ABB RAPID module: ProgSide1.mod

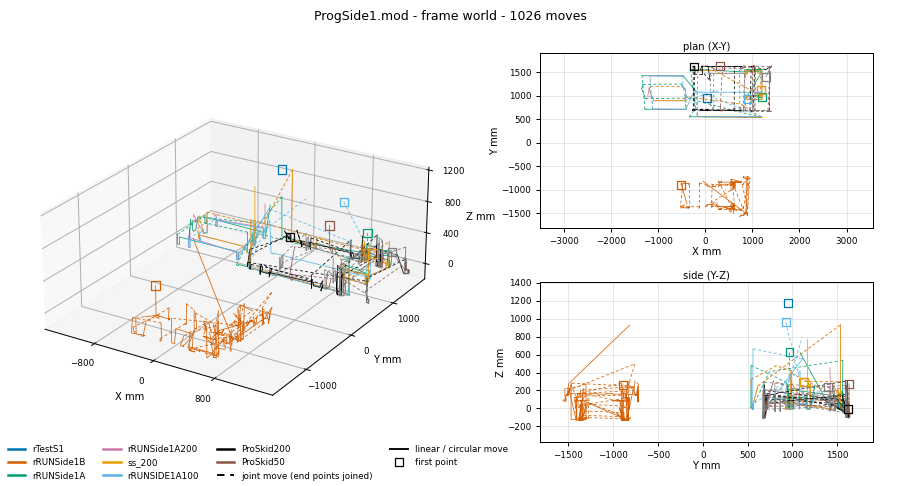
[picture p0: tool path of ProgSide1.mod in frame world, 1026 of 1039 moves have a stored position in this frame; points joined in program order, loops and branches not executed]
MODULE ProgSide1
	PERS bool bZ_B_onlySide2:=FALSE;
	PERS bool bZ_B_onlySide1:=FALSE;
	PERS bool bC_HalfstepSide2:=FALSE;
	PERS bool bC_HalfstepSide1:=FALSE;
	PERS bool bZ_HalfstepSide1:=FALSE;
	PERS bool bZ_HalfstepSide2:=FALSE;
	PERS bool bAngleSide1:=FALSE;
	PERS bool bAngleSide2:=FALSE;
	PERS bool bTestWeldSide1:=FALSE;
    PERS bool bTestWeldSide2:=FALSE;

    ! Boolian initialization for the SS 300 Frames
    PERS bool bNoPartSide1:=FALSE;
	PERS bool bNoPartSide2:=FALSE;
    PERS bool A_onlySide2:=FALSE;
    PERS bool B_onlySide2:=FALSE;
	PERS bool A_onlySide1:=FALSE;
    PERS bool B_onlySide1:=TRUE;
	PERS bool AB_Side1:=FALSE;
    PERS bool AB_Side2:=FALSE;

    ! Boolian initialization for the SelFrames procedures except the SS 300s.
    PERS bool bSkid50:=FALSE;
   	PERS bool bSkid100:=FALSE;
	PERS bool bSkid200:=FALSE;
    PERS bool bSide1A100:=FALSE;
    PERS bool bSide1A200:=FALSE;

    PERS bool bRover:=TRUE;


	TASK PERS welddata weld7:=[15.24,16.6963,[7,0,0,0,0,0,0,0,0],[7,0,0,0,0,0,0,0,0]];
	TASK PERS welddata weld6:=[16.2983,16.6963,[6,0,0,0,0,0,0,0,0],[6,0,0,0,0,0,0,0,0]];

	CONST robtarget pPounceOS1:=[[-398.58,690.45,580.22],[0.00101632,0.999968,-0.00455572,0.00645523],[-1,0,-1,0],[9E+09,9E+09,9E+09,9E+09,9E+09,9E+09]];
	CONST robtarget pPounceS21:=[[580.19,77.23,83.43],[0.071601,0.767336,-0.436334,0.464416],[-1,0,-2,0],[9E+09,9E+09,9E+09,9E+09,9E+09,9E+09]];
	TASK PERS seamdata seam2:=[4,1,[1,0,52,74.0833,0,0,0,0,0],0,0,0,0,0,[1,0,48,0,0,0,0,0,0],0.01,0.1,[1,0,48,105.833,0,0,0,0,0],0,0,[0,0,0,0,0,0,0,0,0],1];
	TASK PERS seamdata seam10:=[4,1,[1,0,50,80.4333,0,0,0,0,0],0,0,0,0,0,[0,0,0,0,0,0,0,0,0],0.25,0.25,[1,0,50,38.1,0,0,0,0,0],0,0,[0,0,0,0,0,0,0,0,0],1];
	CONST robtarget pPounceS31:=[[358.52,159.10,437.93],[0.0181628,-0.398765,0.916866,0.00362624],[-2,0,-2,0],[9E+09,9E+09,9E+09,9E+09,9E+09,9E+09]];
	CONST robtarget pPounceS41:=[[193.25,136.11,113.74],[0.188325,0.84715,-0.195157,0.45693],[-1,-1,-2,0],[9E+09,9E+09,9E+09,9E+09,9E+09,9E+09]];
	PERS welddata weld11:=[13.5467,0,[1,0,50,84.6667,0,0,0,0,0],[0,0,0,0,0,0,0,0,0]];
	PERS welddata weld10:=[14.8167,0,[1,0,50,95.25,0,0,0,0,0],[0,0,0,0,0,0,0,0,0]];
	TASK PERS seamdata seam11:=[1,1,[1,0,50,84.6667,0,0,0,0,0],0,0,0,0,0,[0,0,0,0,0,0,0,0,0],0,0,[0,0,0,0,0,0,0,0,0],0,0,[0,0,0,0,0,0,0,0,0],0];
	TASK PERS seamdata seam12:=[1,1,[1,0,18.5,381,0,0,0,0,0],0,0,0,0,0,[0,0,0,0,0,0,0,0,0],0,0,[0,0,0,0,0,0,0,0,0],0,0,[0,0,0,0,0,0,0,0,0],0];
	TASK PERS seamdata seam13:=[1,1,[1,0,14,127,0,0,0,0,0],0,0,0,0,0,[0,0,0,0,0,0,0,0,0],0,0,[0,0,0,0,0,0,0,0,0],0,0,[0,0,0,0,0,0,0,0,0],0];
	PERS welddata weld12:=[13.97,0,[1,0,50,84.6667,0,0,0,0,0],[0,0,0,0,0,0,0,0,0]];
	PERS welddata weld13:=[6.90033,0,[1,0,20,100.753,0,0,0,0,0],[0,0,0,0,0,0,0,0,0]];
	CONST robtarget pSafeS11:=[[-996.19,963.00,488.78],[0.0459907,-0.688393,0.722625,0.0425673],[1,-1,1,0],[9E+09,9E+09,9E+09,9E+09,9E+09,9E+09]];
	CONST robtarget pSafeS21:=[[-996.19,963.00,488.76],[0.0459983,-0.688397,0.722622,0.0425559],[1,-1,1,0],[9E+09,9E+09,9E+09,9E+09,9E+09,9E+09]];
	CONST robtarget pSafeS31:=[[506.44,675.04,711.34],[0.0314656,-0.935633,0.203865,-0.286426],[0,0,-2,0],[9E+09,9E+09,9E+09,9E+09,9E+09,9E+09]];
	CONST robtarget pSafeS41:=[[488.47,1091.24,654.25],[0.0459806,-0.688392,0.722627,0.0425664],[0,0,-1,0],[9E+09,9E+09,9E+09,9E+09,9E+09,9E+09]];
	CONST robtarget pSafeS51:=[[528.23,1196.89,528.24],[0.224235,-0.753625,-0.525201,-0.325471],[0,-1,-3,0],[9E+09,9E+09,9E+09,9E+09,9E+09,9E+09]];
	CONST robtarget pSafeS61:=[[597.29,1295.03,43.37],[0.191334,-0.732058,-0.538062,-0.371444],[0,-1,-2,0],[9E+09,9E+09,9E+09,9E+09,9E+09,9E+09]];
	CONST robtarget pSafeS71:=[[542.66,1322.39,535.75],[0.223485,-0.764556,-0.487458,-0.357621],[0,-1,-2,0],[9E+09,9E+09,9E+09,9E+09,9E+09,9E+09]];
	CONST robtarget pSafeS81:=[[542.66,1322.38,535.76],[0.223484,-0.764558,-0.487457,-0.35762],[0,-1,-2,0],[9E+09,9E+09,9E+09,9E+09,9E+09,9E+09]];
	CONST robtarget pPounceS51:=[[15.28,993.81,754.75],[0.277209,0.263034,-0.848831,-0.365313],[0,0,0,0],[9E+09,9E+09,9E+09,9E+09,9E+09,9E+09]];
	CONST robtarget pPounceS61:=[[649.55,1131.56,389.19],[0.45355,-0.00505177,-0.879595,-0.143459],[0,0,0,0],[9E+09,9E+09,9E+09,9E+09,9E+09,9E+09]];
	TASK PERS seamdata seam3:=[1,1,[1,0,35,84.6667,0,0,0,0,0],0,0,0,0,0,[1,0,48,0,0,0,0,0,0],0.01,0.1,[1,0,48,105.833,0,0,0,0,0],0,0,[0,0,0,0,0,0,0,0,0],1];
	CONST robtarget pSafeS101:=[[572.94,23.46,738.68],[0.0502756,-0.467207,-0.815726,-0.337314],[0,0,0,0],[9E+09,9E+09,9E+09,9E+09,9E+09,9E+09]];
	CONST robtarget pSafeS111:=[[877.74,-1.14,1156.39],[0.00629855,0.0017594,0.999979,-0.000494623],[0,-1,0,0],[9E+09,9E+09,9E+09,9E+09,9E+09,9E+09]];
	CONST robtarget pSafeS121:=[[877.74,-1.14,1156.39],[0.00629925,0.00175887,0.999979,-0.000492925],[0,-1,0,0],[9E+09,9E+09,9E+09,9E+09,9E+09,9E+09]];
	CONST robtarget pSafeS131:=[[865.02,1139.54,-19.77],[0.144708,-0.274627,0.931028,0.191903],[0,-2,2,0],[9E+09,9E+09,9E+09,9E+09,9E+09,9E+09]];
	CONST robtarget pSafeS141:=[[849.60,1148.97,-24.06],[0.00628216,0.00187497,0.999979,-0.000396021],[0,-1,1,0],[9E+09,9E+09,9E+09,9E+09,9E+09,9E+09]];
	CONST robtarget pSafeS151:=[[1007.97,1505.52,122.27],[0.0460025,-0.688387,0.722632,0.0425454],[0,1,-2,0],[9E+09,9E+09,9E+09,9E+09,9E+09,9E+09]];
	CONST robtarget pHomePos20:=[[365.14,988.92,-33.91],[0.0351389,-0.509982,-0.859022,-0.0276858],[0,-1,1,0],[9E+09,9E+09,9E+09,9E+09,9E+09,9E+09]];
	CONST robtarget pHomePos30:=[[365.15,979.87,-33.91],[0.0351433,-0.509968,-0.85903,-0.0276827],[0,-1,1,0],[9E+09,9E+09,9E+09,9E+09,9E+09,9E+09]];
	CONST robtarget pHomePos40:=[[365.14,979.87,-15.16],[0.0351385,-0.509986,-0.859019,-0.0276867],[0,-1,1,0],[9E+09,9E+09,9E+09,9E+09,9E+09,9E+09]];
	CONST robtarget pHomePos50:=[[433.12,979.73,-15.17],[0.0351369,-0.509964,-0.859032,-0.0276871],[0,-1,1,0],[9E+09,9E+09,9E+09,9E+09,9E+09,9E+09]];
	CONST robtarget pHomePos60:=[[430.57,978.47,-32.25],[0.0351433,-0.50998,-0.859023,-0.0276796],[0,-1,1,0],[9E+09,9E+09,9E+09,9E+09,9E+09,9E+09]];
	CONST robtarget pHomePos70:=[[430.57,978.46,-32.26],[0.0351393,-0.509989,-0.859017,-0.027681],[0,-1,1,0],[9E+09,9E+09,9E+09,9E+09,9E+09,9E+09]];
	CONST robtarget pHomePos80:=[[430.59,974.37,-32.26],[0.0351321,-0.50997,-0.859029,-0.0276862],[0,-1,1,0],[9E+09,9E+09,9E+09,9E+09,9E+09,9E+09]];
	CONST robtarget pHomePos90:=[[430.57,974.36,-24.94],[0.0351397,-0.509992,-0.859016,-0.0276799],[0,-1,1,0],[9E+09,9E+09,9E+09,9E+09,9E+09,9E+09]];
	CONST robtarget pHomePos100:=[[445.83,974.38,-24.94],[0.0351383,-0.509986,-0.859019,-0.0276863],[0,-1,1,0],[9E+09,9E+09,9E+09,9E+09,9E+09,9E+09]];
	CONST robtarget pHomePos110:=[[446.40,974.36,-32.29],[0.0351532,-0.510006,-0.859007,-0.0276708],[0,-1,1,0],[9E+09,9E+09,9E+09,9E+09,9E+09,9E+09]];
	CONST robtarget pHomePos120:=[[446.42,974.37,-32.29],[0.0351424,-0.509994,-0.859014,-0.0276814],[0,-1,1,0],[9E+09,9E+09,9E+09,9E+09,9E+09,9E+09]];
	CONST robtarget pSafeS12:=[[1424.79,-683.57,-13.74],[0.019551,0.168491,0.985501,-0.00412114],[-1,1,-2,0],[9E+09,9E+09,9E+09,9E+09,9E+09,9E+09]];
	CONST robtarget pSafeS22:=[[1462.93,-789.47,-110.40],[0.0637154,0.393325,0.863983,0.307846],[-1,1,-2,0],[9E+09,9E+09,9E+09,9E+09,9E+09,9E+09]];
	CONST robtarget pSafeS32:=[[1462.93,-821.54,-110.39],[0.0637158,0.39332,0.863986,0.307843],[-1,1,-2,0],[9E+09,9E+09,9E+09,9E+09,9E+09,9E+09]];
	CONST robtarget pSafeS42:=[[1462.93,-821.54,-110.39],[0.0637186,0.393326,0.863982,0.307849],[-1,1,-2,0],[9E+09,9E+09,9E+09,9E+09,9E+09,9E+09]];
	CONST robtarget pSafeS52:=[[1462.55,-1477.98,-107.56],[0.0637139,0.393324,0.863983,0.30785],[-1,0,-1,0],[9E+09,9E+09,9E+09,9E+09,9E+09,9E+09]];
	CONST robtarget pSafeS62:=[[1462.54,-1515.56,-107.57],[0.0637098,0.393325,0.863984,0.307846],[-1,0,-1,0],[9E+09,9E+09,9E+09,9E+09,9E+09,9E+09]];
	CONST robtarget pSafeS72:=[[1462.54,-1515.57,-107.57],[0.0637139,0.39333,0.86398,0.307849],[-1,0,-1,0],[9E+09,9E+09,9E+09,9E+09,9E+09,9E+09]];
	CONST robtarget pSafeS82:=[[1462.55,-1515.57,-6.77],[0.063723,0.393334,0.863975,0.307857],[-1,0,-1,0],[9E+09,9E+09,9E+09,9E+09,9E+09,9E+09]];
	CONST robtarget pSafeS161:=[[44.14,948.66,1172.82],[0.0459836,-0.688397,0.722622,0.0425714],[0,-1,0,0],[9E+09,9E+09,9E+09,9E+09,9E+09,9E+09]];
	CONST robtarget pSafeS171:=[[877.68,-1.12,1156.34],[0.00623811,0.00177345,0.999979,-0.000467886],[0,-1,0,0],[9E+09,9E+09,9E+09,9E+09,9E+09,9E+09]];
	CONST robtarget pSafeS181:=[[1178.99,1129.25,299.25],[0.0635535,0.517233,-0.779104,0.348467],[0,1,-3,1],[9E+09,9E+09,9E+09,9E+09,9E+09,9E+09]];
	CONST robtarget pSafeS191:=[[877.68,-1.12,1156.34],[0.00623811,0.00177268,0.999979,-0.000467882],[0,-1,0,0],[9E+09,9E+09,9E+09,9E+09,9E+09,9E+09]];
	CONST robtarget pSafeS201:=[[631.06,-50.80,790.98],[0.377429,-0.0153459,-0.925903,0.00402947],[-1,-1,-5,0],[9E+09,9E+09,9E+09,9E+09,9E+09,9E+09]];
	CONST robtarget pSafeS211:=[[631.06,-50.80,790.98],[0.377429,-0.0153486,-0.925903,0.00403031],[-1,-1,-5,0],[9E+09,9E+09,9E+09,9E+09,9E+09,9E+09]];


!XXXXXXXXXXXXXXXXXXXXXXXXXXXXXXXXXXXXXXXXXXXXXXXXXXXXXXXXXXXX

!XXXXXXXXXXXXXXXXXXXXXXXXXXXXXXXXXXXXXXXXXXXXXXXXXXXXXXXXXXXX
!xxxxxxxxxxxxxxxxxxxxxxxxxxxxxxxxxxxxxxxxxxxxxxxxxxxxxxxxxxxxxxxx




	PROC rNoPartS1()
		MoveJ pSafeS1, v800, fine, tWeldGun;
		MoveJ pPounceS1, v800, fine, tWeldGun;
		MoveJ pSafeS1, v800, fine, tWeldGun;
	ENDPROC
	PROC rTstA1()
		TPWrite "A S1";
	ENDPROC
	PROC rTstB1()
		TPWrite "B S1";
	ENDPROC
	PROC rTestS1()
		MoveJ [[44.14,948.66,1172.81],[0.0459874,-0.688394,0.722625,0.042569],[0,-1,0,0],[9E+09,9E+09,9E+09,9E+09,9E+09,9E+09]], v1000, z50, tWeldGun;
	ENDPROC
	PROC rRUNSide1B()
		rTestPosTop;
		TPWrite "Side 1 B";
		MoveJ [[-516.56,-891.88,262.76],[0.200577,-0.67934,-0.672798,-0.213563],[-2,0,-1,0],[9E+09,9E+09,9E+09,9E+09,9E+09,9E+09]], vmax, z10, tWeldGun;
		MoveL [[-517.38,-892.62,-126.02],[0.230166,-0.665805,-0.672085,-0.228101],[-2,0,-1,0],[9E+09,9E+09,9E+09,9E+09,9E+09,9E+09]], vmax, z10, tWeldGun;
		ArcLStart [[-517.38,-892.61,-138.56],[0.230168,-0.665801,-0.672089,-0.228098],[-2,0,-1,0],[9E+09,9E+09,9E+09,9E+09,9E+09,9E+09]], v50, seam13, weld13\Weave:=weave1, fine, tWeldGun;
		ArcLEnd [[-476.92,-892.72,-138.98],[0.230189,-0.665788,-0.672096,-0.228095],[-2,0,-1,0],[9E+09,9E+09,9E+09,9E+09,9E+09,9E+09]], v10, seam13, weld13\Weave:=weave1, fine, tWeldGun;
		MoveL [[-479.64,-891.87,-91.90],[0.200495,-0.679391,-0.672743,-0.213649],[-2,0,-1,0],[9E+09,9E+09,9E+09,9E+09,9E+09,9E+09]], vmax, z10, tWeldGun;
		MoveJ [[-526.59,-1340.74,-77.97],[0.272049,0.539222,-0.749573,0.270868],[-2,0,-3,0],[9E+09,9E+09,9E+09,9E+09,9E+09,9E+09]], vmax, z10, tWeldGun;
		MoveL [[-521.14,-1337.42,-124.98],[0.179758,0.684801,-0.680481,0.188893],[-2,-1,-3,0],[9E+09,9E+09,9E+09,9E+09,9E+09,9E+09]], vmax, z10, tWeldGun;
		ArcLStart [[-521.16,-1338.85,-130.75],[0.17975,0.684814,-0.680473,0.188882],[-2,-1,-3,0],[9E+09,9E+09,9E+09,9E+09,9E+09,9E+09]], v50, seam13, weld13\Weave:=weave1, fine, tWeldGun;
		ArcLEnd [[-484.70,-1342.96,-133.79],[0.179944,0.684785,-0.680418,0.189003],[-2,-1,-3,0],[9E+09,9E+09,9E+09,9E+09,9E+09,9E+09]], v10, seam13, weld13\Weave:=weave1, fine, tWeldGun;
		MoveL [[-484.84,-1342.71,46.50],[0.235633,0.655478,-0.679432,0.230648],[-2,-1,-3,0],[9E+09,9E+09,9E+09,9E+09,9E+09,9E+09]], vmax, z10, tWeldGun;
		MoveJ [[-392.56,-1296.67,69.52],[0.264192,0.731229,-0.303703,0.550702],[-2,0,0,0],[9E+09,9E+09,9E+09,9E+09,9E+09,9E+09]], vmax, z20, tWeldGun;
		MoveL [[-515.17,-856.60,-124.69],[0.238873,-0.653058,-0.67368,-0.250222],[-2,0,-1,0],[9E+09,9E+09,9E+09,9E+09,9E+09,9E+09]], vmax, z10, tWeldGun;
		ArcLStart [[-515.25,-854.21,-136.09],[0.220515,-0.671496,-0.67216,-0.220606],[-2,0,-1,0],[9E+09,9E+09,9E+09,9E+09,9E+09,9E+09]], v50, seam13, weld13, fine, tWeldGun;
		ArcLEnd [[-491.63,-854.12,-136.10],[0.220508,-0.671473,-0.67215,-0.220715],[-2,0,-1,0],[9E+09,9E+09,9E+09,9E+09,9E+09,9E+09]], v10, seam13, weld13\Weave:=weave1, fine, tWeldGun;
		MoveL [[-479.17,-861.28,-125.34],[0.171406,-0.677441,-0.683701,-0.210352],[-2,0,-1,0],[9E+09,9E+09,9E+09,9E+09,9E+09,9E+09]], vmax, z10, tWeldGun;
		MoveL [[-449.80,-861.68,-125.35],[0.171396,-0.677467,-0.683674,-0.21036],[-2,0,-1,0],[9E+09,9E+09,9E+09,9E+09,9E+09,9E+09]], vmax, z10, tWeldGun;
		ArcLStart [[-449.78,-856.11,-135.93],[0.208269,-0.667838,-0.686513,-0.198285],[-2,0,-1,0],[9E+09,9E+09,9E+09,9E+09,9E+09,9E+09]], v50, seam13, weld13\Weave:=weave1, fine, tWeldGun;
		ArcLEnd [[-419.12,-855.94,-135.97],[0.208222,-0.667816,-0.686496,-0.19847],[-2,0,-1,0],[9E+09,9E+09,9E+09,9E+09,9E+09,9E+09]], v10, seam13, weld13\Weave:=weave1, fine, tWeldGun;
		MoveL [[-410.60,-862.00,-128.92],[0.171386,-0.677508,-0.683632,-0.210375],[-2,0,-1,0],[9E+09,9E+09,9E+09,9E+09,9E+09,9E+09]], vmax, z10, tWeldGun;
		MoveL [[-376.40,-861.00,-128.93],[0.171385,-0.677516,-0.683626,-0.210371],[-2,0,-1,0],[9E+09,9E+09,9E+09,9E+09,9E+09,9E+09]], vmax, z10, tWeldGun;
		ArcLStart [[-376.97,-857.17,-135.72],[0.228827,-0.659649,-0.695979,-0.167674],[-2,0,-1,0],[9E+09,9E+09,9E+09,9E+09,9E+09,9E+09]], v50, seam13, weld13\Weave:=weave1, fine, tWeldGun;
		ArcLEnd [[-359.77,-857.10,-135.74],[0.228871,-0.659593,-0.696016,-0.167683],[-2,0,-1,0],[9E+09,9E+09,9E+09,9E+09,9E+09,9E+09]], v10, seam13, weld13\Weave:=weave1, fine, tWeldGun;
		MoveL [[-340.47,-873.25,-110.32],[0.171334,-0.677678,-0.683442,-0.210489],[-2,0,-1,0],[9E+09,9E+09,9E+09,9E+09,9E+09,9E+09]], vmax, z10, tWeldGun;
		!MoveJ [[-345.72,-887.43,-115.42],[0.0676146,-0.661673,-0.620705,-0.415143],[-2,0,-1,0],[9E+09,9E+09,9E+09,9E+09,9E+09,9E+09]], vmax, z10, tWeldGun;
		!MoveL [[-322.60,-865.30,-126.49],[0.067604,-0.661652,-0.620714,-0.415164],[-2,0,-1,0],[9E+09,9E+09,9E+09,9E+09,9E+09,9E+09]], vmax, z10, tWeldGun;
		!ArcLStart [[-323.53,-854.81,-126.59],[0.0676064,-0.661658,-0.620722,-0.415143],[-2,0,-1,0],[9E+09,9E+09,9E+09,9E+09,9E+09,9E+09]], v50, seam13, weld13, fine, tWeldGun;
		!ArcLEnd [[-310.94,-855.73,-127.27],[0.0675903,-0.661679,-0.620697,-0.415148],[-2,0,-1,0],[9E+09,9E+09,9E+09,9E+09,9E+09,9E+09]], v10, seam13, weld13, fine, tWeldGun;
		MoveL [[-354.07,-859.41,-129.42],[0.135806,-0.859729,-0.404621,-0.280545],[-2,-1,0,0],[9E+09,9E+09,9E+09,9E+09,9E+09,9E+09]], v100, z10, tWeldGun;
		ArcLStart [[-355.40,-857.25,-133.26],[0.101564,-0.865155,-0.372617,-0.319921],[-2,0,0,0],[9E+09,9E+09,9E+09,9E+09,9E+09,9E+09]], v10, seam13, weld13\Weave:=weave1, fine, tWeldGun;
		ArcLEnd [[-352.88,-886.23,-133.63],[0.0471147,-0.867186,-0.374018,-0.325392],[-2,0,-1,0],[9E+09,9E+09,9E+09,9E+09,9E+09,9E+09]], v10, seam13, weld13\Weave:=weave1, fine, tWeldGun;
		MoveL [[-337.59,-890.13,27.38],[0.0676709,-0.661709,-0.620708,-0.415072],[-2,0,-1,0],[9E+09,9E+09,9E+09,9E+09,9E+09,9E+09]], vmax, z10, tWeldGun;
		MoveJ [[-332.34,-1363.85,48.88],[0.219066,0.836756,-0.390875,0.31475],[-2,-1,1,0],[9E+09,9E+09,9E+09,9E+09,9E+09,9E+09]], vmax, z10, tWeldGun;
		MoveL [[-363.40,-1379.69,-125.19],[0.219062,0.836755,-0.390865,0.314767],[-2,-1,1,0],[9E+09,9E+09,9E+09,9E+09,9E+09,9E+09]], vmax, z10, tWeldGun;
		ArcLStart [[-360.34,-1385.64,-128.22],[0.219027,0.836785,-0.39084,0.314741],[-2,-1,1,0],[9E+09,9E+09,9E+09,9E+09,9E+09,9E+09]], v50, seam13, weld13\Weave:=weave1, fine, tWeldGun;
		ArcLEnd [[-360.74,-1353.82,-130.03],[0.219006,0.836811,-0.390806,0.314731],[-2,-1,1,0],[9E+09,9E+09,9E+09,9E+09,9E+09,9E+09]], v10, seam13, weld13\Weave:=weave1, fine, tWeldGun;
		MoveL [[-339.52,-1381.52,-122.91],[0.192161,0.836468,-0.399943,0.321625],[-2,-1,1,0],[9E+09,9E+09,9E+09,9E+09,9E+09,9E+09]], vmax, z10, tWeldGun;
		MoveL [[-360.99,-1380.78,-119.54],[0.218983,0.836818,-0.390808,0.314725],[-2,-1,1,0],[9E+09,9E+09,9E+09,9E+09,9E+09,9E+09]], vmax, z10, tWeldGun;
		ArcLStart [[-361.02,-1385.20,-130.65],[0.211582,0.836718,-0.393407,0.316807],[-2,-1,1,0],[9E+09,9E+09,9E+09,9E+09,9E+09,9E+09]], v10, seam13, weld13\Weave:=weave1, fine, tWeldGun;
		ArcLEnd [[-390.01,-1385.18,-131.66],[0.209306,0.844003,-0.389899,0.303035],[-2,-1,1,0],[9E+09,9E+09,9E+09,9E+09,9E+09,9E+09]], v10, seam13, weld13\Weave:=weave1, fine, tWeldGun;
		MoveL [[-390.07,-1379.88,-124.94],[0.206619,0.84095,-0.396616,0.304645],[-2,-1,1,0],[9E+09,9E+09,9E+09,9E+09,9E+09,9E+09]], vmax, z10, tWeldGun;
		!ArcLStart [[-352.45,-1380.36,-127.77],[0.213181,0.666131,-0.683648,0.208447],[-2,-1,1,0],[9E+09,9E+09,9E+09,9E+09,9E+09,9E+09]], v30, seam13, weld13, fine, tWeldGun;
		!ArcLEnd [[-392.89,-1382.82,-132.94],[0.213455,0.666087,-0.683527,0.208703],[-2,-1,1,0],[9E+09,9E+09,9E+09,9E+09,9E+09,9E+09]], v10, seam13, weld13, fine, tWeldGun;
		MoveL [[-383.12,-1377.19,-116.87],[0.247825,0.654497,-0.670463,0.246367],[-2,-1,1,0],[9E+09,9E+09,9E+09,9E+09,9E+09,9E+09]], vmax, z10, tWeldGun;
		MoveL [[-423.74,-1380.30,-127.27],[0.236796,0.658364,-0.678163,0.2249],[-2,-1,1,0],[9E+09,9E+09,9E+09,9E+09,9E+09,9E+09]], vmax, z10, tWeldGun;
		ArcLStart [[-423.76,-1381.10,-131.68],[0.205145,0.668814,-0.684061,0.206555],[-2,-1,1,0],[9E+09,9E+09,9E+09,9E+09,9E+09,9E+09]], v50, seam13, weld13\Weave:=weave1, fine, tWeldGun;
		ArcLEnd [[-450.34,-1381.29,-131.68],[0.205213,0.668788,-0.684058,0.206581],[-2,-1,1,0],[9E+09,9E+09,9E+09,9E+09,9E+09,9E+09]], v10, seam13, weld13\Weave:=weave1, fine, tWeldGun;
		MoveL [[-450.89,-1376.20,-127.31],[0.205227,0.668769,-0.684078,0.20656],[-2,-1,1,0],[9E+09,9E+09,9E+09,9E+09,9E+09,9E+09]], vmax, z10, tWeldGun;
		MoveL [[-485.27,-1373.50,-126.43],[0.24151,0.665828,-0.67086,0.219756],[-2,-1,1,0],[9E+09,9E+09,9E+09,9E+09,9E+09,9E+09]], vmax, z10, tWeldGun;
		ArcLStart [[-485.09,-1381.68,-132.22],[0.234587,0.663654,-0.676661,0.216014],[-2,-1,1,0],[9E+09,9E+09,9E+09,9E+09,9E+09,9E+09]], v50, seam13, weld13\Weave:=weave1, fine, tWeldGun;
		ArcLEnd [[-523.10,-1381.58,-132.24],[0.234599,0.66365,-0.676663,0.216008],[-2,-1,1,0],[9E+09,9E+09,9E+09,9E+09,9E+09,9E+09]], v10, seam13, weld13\Weave:=weave1, fine, tWeldGun;
		MoveL [[-522.10,-1355.74,48.22],[0.158867,0.68146,-0.647455,0.301955],[-2,0,1,0],[9E+09,9E+09,9E+09,9E+09,9E+09,9E+09]], vmax, z10, tWeldGun;
		MoveJ [[-133.27,-1356.80,81.68],[0.311551,0.028851,-0.949681,-0.0145225],[-2,0,-2,0],[9E+09,9E+09,9E+09,9E+09,9E+09,9E+09]], vmax, z10, tWeldGun;
		MoveL [[-129.77,-1359.47,-118.55],[0.313406,-0.0329684,-0.948479,0.032837],[-2,0,-2,0],[9E+09,9E+09,9E+09,9E+09,9E+09,9E+09]], vmax, z10, tWeldGun;
		ArcLStart [[-130.10,-1360.61,-131.11],[0.319988,-0.0412281,-0.946509,0.00534418],[-2,0,-2,0],[9E+09,9E+09,9E+09,9E+09,9E+09,9E+09]], v50, seam13, weld13\Weave:=weave1, fine, tWeldGun;
		ArcLEnd [[-130.29,-1389.82,-131.10],[0.320004,-0.0412218,-0.946504,0.00536126],[-2,0,-2,0],[9E+09,9E+09,9E+09,9E+09,9E+09,9E+09]], v10, seam13, weld13\Weave:=weave1, fine, tWeldGun;
		MoveL [[-127.94,-1387.70,-99.83],[0.311507,0.0288878,-0.94969,-0.0147574],[-2,0,-2,0],[9E+09,9E+09,9E+09,9E+09,9E+09,9E+09]], vmax, z10, tWeldGun;
		MoveJ [[-120.34,-878.23,-115.66],[0.321395,0.00587998,-0.946893,0.00807266],[-2,0,-2,0],[9E+09,9E+09,9E+09,9E+09,9E+09,9E+09]], vmax, z10, tWeldGun;
		MoveL [[-125.84,-880.54,-126.77],[0.319682,0.0182803,-0.947348,-0.00115479],[-2,0,-2,0],[9E+09,9E+09,9E+09,9E+09,9E+09,9E+09]], vmax, z10, tWeldGun;
		ArcLStart [[-127.17,-881.43,-133.73],[0.308264,0.0190236,-0.951103,0.00389985],[-2,0,-2,0],[9E+09,9E+09,9E+09,9E+09,9E+09,9E+09]], v50, seam13, weld13\Weave:=weave1, fine, tWeldGun;
		ArcLEnd [[-126.99,-850.35,-133.72],[0.308286,0.0190346,-0.951095,0.00390381],[-2,0,-2,0],[9E+09,9E+09,9E+09,9E+09,9E+09,9E+09]], v10, seam13, weld13\Weave:=weave1, fine, tWeldGun;
		MoveL [[-126.07,-851.54,117.21],[0.311664,0.0289025,-0.949643,-0.0144782],[-2,0,-2,0],[9E+09,9E+09,9E+09,9E+09,9E+09,9E+09]], vmax, z10, tWeldGun;
		MoveJ [[5.08,-892.16,87.65],[0.246917,-0.649526,-0.670091,-0.261011],[-2,0,-1,0],[9E+09,9E+09,9E+09,9E+09,9E+09,9E+09]], vmax, z10, tWeldGun;
		MoveL [[5.70,-898.13,-125.58],[0.246931,-0.64953,-0.670081,-0.261012],[-2,0,-1,0],[9E+09,9E+09,9E+09,9E+09,9E+09,9E+09]], vmax, z10, tWeldGun;
		ArcLStart [[8.01,-895.77,-137.58],[0.202938,-0.669252,-0.681328,-0.216127],[-2,0,-1,0],[9E+09,9E+09,9E+09,9E+09,9E+09,9E+09]], v50, seam13, weld13\Weave:=weave1, fine, tWeldGun;
		ArcLEnd [[39.00,-896.37,-138.18],[0.202954,-0.669237,-0.681341,-0.216117],[-1,0,-1,0],[9E+09,9E+09,9E+09,9E+09,9E+09,9E+09]], v10, seam13, weld13\Weave:=weave1, fine, tWeldGun;
		MoveL [[40.66,-920.62,70.48],[0.246699,-0.649617,-0.670207,-0.260692],[-1,0,-1,0],[9E+09,9E+09,9E+09,9E+09,9E+09,9E+09]], vmax, z10, tWeldGun;
		MoveJ [[283.83,-931.65,13.13],[0.246958,-0.649486,-0.670134,-0.26096],[-1,0,0,0],[9E+09,9E+09,9E+09,9E+09,9E+09,9E+09]], vmax, z10, tWeldGun;
		MoveL [[286.40,-898.85,-115.99],[0.246961,-0.649476,-0.670147,-0.26095],[-1,0,0,0],[9E+09,9E+09,9E+09,9E+09,9E+09,9E+09]], vmax, z10, tWeldGun;
		ArcLStart [[287.27,-897.40,-138.20],[0.199806,-0.665794,-0.68607,-0.214718],[-1,-1,0,0],[9E+09,9E+09,9E+09,9E+09,9E+09,9E+09]], v50, seam13, weld13\Weave:=weave1, fine, tWeldGun;
		ArcLEnd [[316.06,-898.20,-138.20],[0.19983,-0.665775,-0.686086,-0.214705],[-1,-1,0,0],[9E+09,9E+09,9E+09,9E+09,9E+09,9E+09]], v10, seam13, weld13\Weave:=weave1, fine, tWeldGun;
		MoveL [[299.75,-898.83,-116.82],[0.246966,-0.649478,-0.670145,-0.260945],[-1,0,0,0],[9E+09,9E+09,9E+09,9E+09,9E+09,9E+09]], vmax, z10, tWeldGun;
		MoveJ [[559.57,-898.83,-116.82],[0.246966,-0.649476,-0.670148,-0.260944],[-1,-1,0,0],[9E+09,9E+09,9E+09,9E+09,9E+09,9E+09]], vmax, z10, tWeldGun;
		MoveL [[564.80,-902.55,-126.00],[0.209407,-0.662689,-0.684007,-0.221648],[-1,-1,0,0],[9E+09,9E+09,9E+09,9E+09,9E+09,9E+09]], vmax, z10, tWeldGun;
		ArcLStart [[567.30,-900.67,-135.77],[0.209518,-0.662633,-0.684042,-0.221601],[-1,-1,0,0],[9E+09,9E+09,9E+09,9E+09,9E+09,9E+09]], v50, seam13, weld13\Weave:=weave1, fine, tWeldGun;
		ArcLEnd [[598.83,-900.83,-136.39],[0.209539,-0.662615,-0.684059,-0.221582],[-1,-1,0,0],[9E+09,9E+09,9E+09,9E+09,9E+09,9E+09]], v10, seam13, weld13\Weave:=weave1, fine, tWeldGun;
		MoveL [[596.75,-960.43,-56.34],[0.246991,-0.649449,-0.670174,-0.260919],[-1,-1,0,0],[9E+09,9E+09,9E+09,9E+09,9E+09,9E+09]], vmax, z10, tWeldGun;
		MoveJ [[601.90,-897.43,-123.32],[0.32616,-0.613254,-0.630335,-0.346725],[-1,0,0,0],[9E+09,9E+09,9E+09,9E+09,9E+09,9E+09]], vmax, z10, tWeldGun;
		MoveL [[600.91,-903.21,-128.01],[0.274675,-0.639039,-0.654325,-0.296719],[-1,0,0,0],[9E+09,9E+09,9E+09,9E+09,9E+09,9E+09]], v100, z10, tWeldGun;
		ArcLStart [[600.91,-897.21,-134.81],[0.274671,-0.63904,-0.654325,-0.296721],[-1,0,0,0],[9E+09,9E+09,9E+09,9E+09,9E+09,9E+09]], v10, seam13, weld13\Weave:=weave1, fine, tWeldGun;
		ArcLEnd [[631.68,-897.21,-134.82],[0.274687,-0.639035,-0.654325,-0.296718],[-1,0,0,0],[9E+09,9E+09,9E+09,9E+09,9E+09,9E+09]], v10, seam13, weld13\Weave:=weave1, fine, tWeldGun;
		MoveL [[633.74,-910.04,-132.93],[0.326202,-0.613258,-0.630325,-0.346695],[-1,0,0,0],[9E+09,9E+09,9E+09,9E+09,9E+09,9E+09]], vmax, z10, tWeldGun;
		MoveL [[633.73,-910.04,183.03],[0.326216,-0.613247,-0.630334,-0.346685],[-1,0,0,0],[9E+09,9E+09,9E+09,9E+09,9E+09,9E+09]], vmax, z10, tWeldGun;
		MoveJ [[627.00,-822.44,298.30],[0.361159,0.600904,-0.609737,0.36973],[-1,-1,-2,0],[9E+09,9E+09,9E+09,9E+09,9E+09,9E+09]], vmax, z10, tWeldGun;
		MoveL [[626.21,-835.86,-135.39],[0.402337,0.574507,-0.586331,0.405317],[-1,-2,-1,0],[9E+09,9E+09,9E+09,9E+09,9E+09,9E+09]], vmax, z10, tWeldGun;
		ArcLStart [[627.33,-853.89,-136.93],[0.402422,0.574444,-0.586338,0.405314],[-1,-2,-1,0],[9E+09,9E+09,9E+09,9E+09,9E+09,9E+09]], v50, seam13, weld13\Weave:=weave1, fine, tWeldGun;
		ArcLEnd [[595.13,-853.88,-136.75],[0.402409,0.574476,-0.586313,0.405318],[-1,-2,-1,0],[9E+09,9E+09,9E+09,9E+09,9E+09,9E+09]], v10, seam13, weld13\Weave:=weave1, fine, tWeldGun;
		MoveL [[595.98,-827.09,-135.34],[0.402393,0.574513,-0.586267,0.405347],[-1,-2,-1,0],[9E+09,9E+09,9E+09,9E+09,9E+09,9E+09]], vmax, z10, tWeldGun;
		MoveL [[626.55,-840.41,83.52],[0.487695,0.50329,-0.532941,0.47416],[-1,-2,-1,0],[9E+09,9E+09,9E+09,9E+09,9E+09,9E+09]], vmax, z10, tWeldGun;
		!MoveJ [[591.71,-1338.72,-121.22],[0.313919,0.593482,-0.705938,0.225579],[-1,-1,2,0],[9E+09,9E+09,9E+09,9E+09,9E+09,9E+09]], v1000, z10, tWeldGun;
		!MoveL [[591.71,-1350.59,-131.13],[0.31392,0.593478,-0.705939,0.225584],[-1,-1,2,0],[9E+09,9E+09,9E+09,9E+09,9E+09,9E+09]], v1000, z10, tWeldGun;
		ArcLStart [[627.59,-855.49,80.83],[0.48302,0.507656,-0.528665,0.479052],[-1,-2,-1,0],[9E+09,9E+09,9E+09,9E+09,9E+09,9E+09]], v40, seam13, weld13\Weave:=weave1, fine, tWeldGun;
		ArcLEnd [[594.18,-855.46,80.81],[0.483027,0.507675,-0.528656,0.479035],[-1,-2,-1,0],[9E+09,9E+09,9E+09,9E+09,9E+09,9E+09]], v10, seam13, weld13\Weave:=weave1, fine, tWeldGun;
		MoveL [[594.80,-840.42,83.53],[0.487698,0.503251,-0.532984,0.47415],[-1,-2,-1,0],[9E+09,9E+09,9E+09,9E+09,9E+09,9E+09]], vmax, z10, tWeldGun;
		SingArea\Wrist;
		MoveJ [[510.38,-859.01,160.69],[0.00485322,0.746032,-0.024255,0.665452],[-1,0,0,0],[9E+09,9E+09,9E+09,9E+09,9E+09,9E+09]], vmax, z10, tWeldGun;
		MoveL [[594.98,-857.13,82.26],[0.0048321,0.745919,-0.0242101,0.665579],[-1,0,0,0],[9E+09,9E+09,9E+09,9E+09,9E+09,9E+09]], vmax, z10, tWeldGun;
		ArcLStart [[600.76,-855.94,81.47],[0.00483992,0.74593,-0.0242017,0.665567],[-1,0,0,0],[9E+09,9E+09,9E+09,9E+09,9E+09,9E+09]], v40, seam13, weld13\Weave:=weave1, fine, tWeldGun;
		ArcLEnd [[600.72,-888.35,80.66],[0.00484822,0.745947,-0.0241951,0.665549],[-1,0,0,0],[9E+09,9E+09,9E+09,9E+09,9E+09,9E+09]], v10, seam13, weld13\Weave:=weave1, fine, tWeldGun;
		MoveL [[545.64,-889.59,83.73],[0.0047987,0.745982,-0.0242261,0.665508],[-1,0,0,0],[9E+09,9E+09,9E+09,9E+09,9E+09,9E+09]], vmax, z10, tWeldGun;
		MoveL [[545.47,-1007.73,83.69],[0.00477345,0.745999,-0.0242032,0.665491],[-1,0,0,0],[9E+09,9E+09,9E+09,9E+09,9E+09,9E+09]], vmax, z10, tWeldGun;
		MoveJ [[631.13,-962.99,83.64],[0.467638,-0.538268,-0.512971,-0.477958],[-1,0,0,0],[9E+09,9E+09,9E+09,9E+09,9E+09,9E+09]], vmax, z10, tWeldGun;
		MoveL [[598.81,-898.79,83.47],[0.467222,-0.531735,-0.519712,-0.478395],[-1,0,0,0],[9E+09,9E+09,9E+09,9E+09,9E+09,9E+09]], vmax, z10, tWeldGun;
		ArcLStart [[601.50,-884.14,82.85],[0.46721,-0.531727,-0.519721,-0.478406],[-1,0,0,0],[9E+09,9E+09,9E+09,9E+09,9E+09,9E+09]], v50, seam13, weld13\Weave:=weave1, fine, tWeldGun;
		ArcLEnd [[633.51,-883.86,83.69],[0.46722,-0.531721,-0.519715,-0.478409],[-1,0,0,0],[9E+09,9E+09,9E+09,9E+09,9E+09,9E+09]], v10, seam13, weld13\Weave:=weave1, fine, tWeldGun;
		MoveL [[633.84,-953.29,84.81],[0.467086,-0.531839,-0.51974,-0.478381],[-1,0,0,0],[9E+09,9E+09,9E+09,9E+09,9E+09,9E+09]], vmax, z10, tWeldGun;
		MoveJ [[-0.34,-1346.80,171.20],[0.287604,0.644423,-0.651566,0.278325],[-1,-1,-2,0],[9E+09,9E+09,9E+09,9E+09,9E+09,9E+09]], vmax, z10, tWeldGun;
		MoveL [[-2.12,-1347.00,-106.57],[0.287602,0.644471,-0.651521,0.278323],[-1,-1,-2,0],[9E+09,9E+09,9E+09,9E+09,9E+09,9E+09]], vmax, z10, tWeldGun;
		ArcLStart [[0.53,-1348.45,-134.66],[0.24536,0.661385,-0.66625,0.241826],[-1,0,-2,0],[9E+09,9E+09,9E+09,9E+09,9E+09,9E+09]], v40, seam13, weld13\Weave:=weave1, fine, tWeldGun;
		ArcLEnd [[35.28,-1348.02,-135.08],[0.245344,0.66148,-0.666161,0.241829],[-1,0,-2,0],[9E+09,9E+09,9E+09,9E+09,9E+09,9E+09]], v10, seam13, weld13\Weave:=weave1, fine, tWeldGun;
		MoveL [[33.45,-1306.76,35.10],[0.287609,0.644475,-0.651512,0.278328],[-1,-1,-2,0],[9E+09,9E+09,9E+09,9E+09,9E+09,9E+09]], vmax, z10, tWeldGun;
		MoveL [[273.41,-1327.02,35.12],[0.287608,0.6445,-0.651487,0.278327],[-1,-1,-2,0],[9E+09,9E+09,9E+09,9E+09,9E+09,9E+09]], vmax, z10, tWeldGun;
		MoveL [[278.63,-1350.36,-113.58],[0.287595,0.644518,-0.651477,0.278323],[-1,-1,-2,0],[9E+09,9E+09,9E+09,9E+09,9E+09,9E+09]], vmax, z10, tWeldGun;
		ArcLStart [[281.41,-1351.07,-135.11],[0.23791,0.664067,-0.669311,0.233317],[-1,0,-2,0],[9E+09,9E+09,9E+09,9E+09,9E+09,9E+09]], v40, seam13, weld13\Weave:=weave1, fine, tWeldGun;
		ArcLEnd [[314.07,-1351.40,-135.14],[0.237905,0.66408,-0.669298,0.233324],[-1,0,-2,0],[9E+09,9E+09,9E+09,9E+09,9E+09,9E+09]], v10, seam13, weld13\Weave:=weave1, fine, tWeldGun;
		MoveL [[313.56,-1350.36,-117.72],[0.287596,0.644518,-0.651477,0.278324],[-1,-1,-2,0],[9E+09,9E+09,9E+09,9E+09,9E+09,9E+09]], vmax, z10, tWeldGun;
		MoveL [[556.08,-1348.76,-117.74],[0.287601,0.644532,-0.651463,0.278317],[-1,-1,-2,0],[9E+09,9E+09,9E+09,9E+09,9E+09,9E+09]], vmax, z10, tWeldGun;
		ArcLStart [[558.44,-1352.44,-134.04],[0.243015,0.662361,-0.668163,0.23618],[-1,0,-2,0],[9E+09,9E+09,9E+09,9E+09,9E+09,9E+09]], v40, seam13, weld13\Weave:=weave1, fine, tWeldGun;
		ArcLEnd [[594.43,-1353.65,-134.07],[0.265401,0.653922,-0.658502,0.26139],[-1,0,-2,0],[9E+09,9E+09,9E+09,9E+09,9E+09,9E+09]], v10, seam13, weld13\Weave:=weave1, fine, tWeldGun;
		MoveL [[591.10,-1294.92,-96.48],[0.287644,0.644544,-0.6514,0.278391],[-1,-1,-2,0],[9E+09,9E+09,9E+09,9E+09,9E+09,9E+09]], vmax, z10, tWeldGun;
		!MoveJ [[629.17,-1265.05,-98.00],[0.340013,0.628245,-0.617658,0.328935],[-1,-1,-2,0],[9E+09,9E+09,9E+09,9E+09,9E+09,9E+09]], vmax, z10, tWeldGun;
		MoveL [[623.54,-1349.21,-127.64],[0.3277,0.635367,-0.623181,0.317123],[-1,-1,-2,0],[9E+09,9E+09,9E+09,9E+09,9E+09,9E+09]], vmax, z10, tWeldGun;
		ArcLStart [[622.97,-1358.18,-133.65],[0.327698,0.635371,-0.623176,0.317128],[-1,-1,-2,0],[9E+09,9E+09,9E+09,9E+09,9E+09,9E+09]], v40, seam13, weld13\Weave:=weave1, fine, tWeldGun;
		ArcLEnd [[591.94,-1357.90,-133.23],[0.327693,0.635344,-0.623186,0.317167],[-1,-1,-2,0],[9E+09,9E+09,9E+09,9E+09,9E+09,9E+09]], v10, seam13, weld13\Weave:=weave1, fine, tWeldGun;
		MoveL [[594.26,-1304.04,-124.90],[0.375061,0.603881,-0.605571,0.35769],[-1,-1,-2,0],[9E+09,9E+09,9E+09,9E+09,9E+09,9E+09]], vmax, z10, tWeldGun;
		MoveL [[594.27,-1304.02,270.29],[0.377187,0.607515,-0.60193,0.355439],[-1,-1,-2,0],[9E+09,9E+09,9E+09,9E+09,9E+09,9E+09]], vmax, z10, tWeldGun;
		MoveJ [[598.90,-1494.47,216.89],[0.17643,-0.701594,-0.668329,-0.173135],[-1,-1,0,0],[9E+09,9E+09,9E+09,9E+09,9E+09,9E+09]], vmax, z10, tWeldGun;
		MoveL [[597.76,-1413.70,-132.21],[0.38046,-0.610425,-0.582563,-0.378488],[-1,0,0,0],[9E+09,9E+09,9E+09,9E+09,9E+09,9E+09]], vmax, z10, tWeldGun;
		ArcLStart [[594.86,-1404.13,-132.25],[0.380476,-0.61045,-0.582552,-0.378447],[-1,0,0,0],[9E+09,9E+09,9E+09,9E+09,9E+09,9E+09]], v50, seam13, weld13\Weave:=weave1, fine, tWeldGun;
		ArcLEnd [[628.57,-1403.11,-132.15],[0.38049,-0.610453,-0.582547,-0.378435],[-1,0,0,0],[9E+09,9E+09,9E+09,9E+09,9E+09,9E+09]], v10, seam13, weld13\Weave:=weave1, fine, tWeldGun;
		MoveL [[628.36,-1412.35,-121.21],[0.467542,-0.524108,-0.539123,-0.464825],[-1,0,0,0],[9E+09,9E+09,9E+09,9E+09,9E+09,9E+09]], vmax, z10, tWeldGun;
		MoveL [[629.51,-1407.41,86.42],[0.467564,-0.524053,-0.539189,-0.464788],[-1,0,0,0],[9E+09,9E+09,9E+09,9E+09,9E+09,9E+09]], vmax, z10, tWeldGun;
		ArcLStart [[628.33,-1394.78,86.06],[0.467613,-0.524083,-0.539148,-0.464753],[-1,0,0,0],[9E+09,9E+09,9E+09,9E+09,9E+09,9E+09]], v40, seam13, weld13\Weave:=weave1, fine, tWeldGun;
		ArcLEnd [[594.53,-1394.77,86.03],[0.467622,-0.524085,-0.539138,-0.464753],[-1,0,0,0],[9E+09,9E+09,9E+09,9E+09,9E+09,9E+09]], v10, seam13, weld13\Weave:=weave1, fine, tWeldGun;
		MoveL [[595.96,-1403.58,86.03],[0.467592,-0.524062,-0.539124,-0.464825],[-1,0,0,0],[9E+09,9E+09,9E+09,9E+09,9E+09,9E+09]], vmax, z10, tWeldGun;
		MoveL [[457.06,-1403.59,89.42],[0.225264,-0.323777,-0.705869,-0.588366],[-1,0,-1,0],[9E+09,9E+09,9E+09,9E+09,9E+09,9E+09]], vmax, z10, tWeldGun;
		MoveJ [[483.55,-1400.78,96.25],[0.150969,0.719954,0.110873,0.668268],[-1,0,0,0],[9E+09,9E+09,9E+09,9E+09,9E+09,9E+09]], vmax, z10, tWeldGun;
		MoveL [[583.47,-1400.75,85.01],[0.0329721,0.73526,0.0213877,0.676645],[-1,0,0,0],[9E+09,9E+09,9E+09,9E+09,9E+09,9E+09]], vmax, z10, tWeldGun;
		ArcLStart [[594.01,-1399.37,84.43],[0.0288105,0.735302,0.0250795,0.676663],[-1,0,0,0],[9E+09,9E+09,9E+09,9E+09,9E+09,9E+09]], v50, seam13, weld13\Weave:=weave1, fine, tWeldGun;
		ArcLEnd [[593.57,-1367.91,84.17],[0.028766,0.73533,0.0251421,0.676632],[-1,0,0,0],[9E+09,9E+09,9E+09,9E+09,9E+09,9E+09]], v10, seam13, weld13\Weave:=weave1, fine, tWeldGun;
		MoveL [[554.18,-1372.28,89.73],[0.15109,0.720146,0.110407,0.668112],[-1,0,0,0],[9E+09,9E+09,9E+09,9E+09,9E+09,9E+09]], vmax, z10, tWeldGun;
		MoveL [[549.71,-1268.25,89.71],[0.151117,0.720151,0.110329,0.668113],[-1,1,0,0],[9E+09,9E+09,9E+09,9E+09,9E+09,9E+09]], vmax, z10, tWeldGun;
		MoveJ [[603.39,-1313.43,143.58],[0.469159,0.533622,-0.523436,0.470269],[-1,-2,3,0],[9E+09,9E+09,9E+09,9E+09,9E+09,9E+09]], vmax, z10, tWeldGun;
		MoveL [[591.28,-1347.97,82.12],[0.473675,0.523571,-0.526883,0.473181],[-1,-2,3,0],[9E+09,9E+09,9E+09,9E+09,9E+09,9E+09]], vmax, z10, tWeldGun;
		ArcLStart [[587.84,-1367.93,83.28],[0.473679,0.523503,-0.526973,0.473152],[-1,-2,3,0],[9E+09,9E+09,9E+09,9E+09,9E+09,9E+09]], v40, seam13, weld13\Weave:=weave1, fine, tWeldGun;
		ArcLEnd [[621.99,-1367.50,82.25],[0.473695,0.523434,-0.527058,0.473118],[-1,-2,3,0],[9E+09,9E+09,9E+09,9E+09,9E+09,9E+09]], v10, seam13, weld13\Weave:=weave1, fine, tWeldGun;
		MoveL [[621.57,-1338.36,83.93],[0.473691,0.523533,-0.526918,0.473168],[-1,-2,3,0],[9E+09,9E+09,9E+09,9E+09,9E+09,9E+09]], vmax, z10, tWeldGun;
		!MoveL [[592.94,-1347.68,-124.63],[0.145068,0.695314,-0.634216,0.305394],[-1,0,1,0],[9E+09,9E+09,9E+09,9E+09,9E+09,9E+09]], vmax, z10, tWeldGun;
		!ArcLStart [[592.95,-1351.62,-131.66],[0.121904,0.705948,-0.639076,0.279928],[-1,0,1,0],[9E+09,9E+09,9E+09,9E+09,9E+09,9E+09]], v40, seam13, weld13\Weave:=weave1, fine, tWeldGun;
		!ArcLEnd [[553.63,-1351.63,-131.65],[0.121904,0.705942,-0.639079,0.279934],[-1,0,1,0],[9E+09,9E+09,9E+09,9E+09,9E+09,9E+09]], v10, seam13, weld13\Weave:=weave1, fine, tWeldGun;
		!MoveL [[558.95,-1354.44,-113.35],[0.145045,0.695254,-0.634278,0.305412],[-1,0,1,0],[9E+09,9E+09,9E+09,9E+09,9E+09,9E+09]], vmax, z10, tWeldGun;
		!MoveL [[313.92,-1351.24,-119.86],[0.226173,0.673271,-0.665892,0.228343],[-1,0,2,0],[9E+09,9E+09,9E+09,9E+09,9E+09,9E+09]], vmax, z10, tWeldGun;
		!ArcLStart [[315.31,-1349.16,-136.09],[0.226124,0.673334,-0.665847,0.228338],[-1,0,2,0],[9E+09,9E+09,9E+09,9E+09,9E+09,9E+09]], v40, seam13, weld13\Weave:=weave1, fine, tWeldGun;
		!ArcLEnd [[277.70,-1348.77,-134.69],[0.226134,0.673338,-0.66584,0.228336],[-1,0,2,0],[9E+09,9E+09,9E+09,9E+09,9E+09,9E+09]], v10, seam13, weld13\Weave:=weave1, fine, tWeldGun;
		!MoveL [[279.11,-1351.10,-105.85],[0.22616,0.673298,-0.665876,0.228321],[-1,0,2,0],[9E+09,9E+09,9E+09,9E+09,9E+09,9E+09]], vmax, z10, tWeldGun;
		MoveJ [[584.48,-948.55,-60.93],[0.252385,-0.649774,-0.664987,-0.268121],[-1,0,0,0],[9E+09,9E+09,9E+09,9E+09,9E+09,9E+09]], vmax, z10, tWeldGun;
		MoveL [[587.25,-889.04,-107.33],[0.252799,-0.649451,-0.665162,-0.268079],[-1,0,0,0],[9E+09,9E+09,9E+09,9E+09,9E+09,9E+09]], vmax, z10, tWeldGun;
		ArcLStart [[587.97,-882.93,-130.55],[0.253029,-0.649357,-0.665187,-0.268027],[-1,0,0,0],[9E+09,9E+09,9E+09,9E+09,9E+09,9E+09]], v40, seam13, weld13\Weave:=weave1, fine, tWeldGun;
		ArcL [[579.89,-891.69,-131.98],[0.25302,-0.649426,-0.665094,-0.2681],[-1,0,0,0],[9E+09,9E+09,9E+09,9E+09,9E+09,9E+09]], v10, seam13, weld13\Weave:=weave1, z0, tWeldGun;
		ArcL [[479.92,-890.95,-132.98],[0.253042,-0.649377,-0.665146,-0.26807],[-1,0,0,0],[9E+09,9E+09,9E+09,9E+09,9E+09,9E+09]], v10, seam13, weld13\Weave:=weave1, z0, tWeldGun;
		ArcLEnd [[469.00,-879.31,-133.61],[0.253095,-0.649334,-0.665183,-0.26803],[-1,0,0,0],[9E+09,9E+09,9E+09,9E+09,9E+09,9E+09]], v10, seam13, weld13\Weave:=weave1, fine, tWeldGun;
		MoveL [[472.59,-879.09,-111.98],[0.253025,-0.6494,-0.665124,-0.268085],[-1,0,0,0],[9E+09,9E+09,9E+09,9E+09,9E+09,9E+09]], vmax, z10, tWeldGun;
		MoveL [[396.83,-879.33,-105.08],[0.253072,-0.649383,-0.665131,-0.268064],[-1,0,0,0],[9E+09,9E+09,9E+09,9E+09,9E+09,9E+09]], vmax, z10, tWeldGun;
		ArcLStart [[396.64,-879.58,-133.89],[0.25962,-0.646746,-0.667845,-0.261344],[-1,-1,0,0],[9E+09,9E+09,9E+09,9E+09,9E+09,9E+09]], v40, seam13, weld13\Weave:=weave1, fine, tWeldGun;
		ArcL [[385.74,-890.30,-133.85],[0.253227,-0.649246,-0.665248,-0.267957],[-1,0,0,0],[9E+09,9E+09,9E+09,9E+09,9E+09,9E+09]], v10, seam13, weld13\Weave:=weave1, z0, tWeldGun;
		ArcLEnd [[339.88,-890.45,-134.28],[0.253187,-0.649517,-0.664897,-0.268209],[-1,0,0,0],[9E+09,9E+09,9E+09,9E+09,9E+09,9E+09]], v10, seam13, weld13\Weave:=weave1, fine, tWeldGun;
		MoveL [[339.91,-888.27,-120.68],[0.253151,-0.649537,-0.664886,-0.268224],[-1,0,0,0],[9E+09,9E+09,9E+09,9E+09,9E+09,9E+09]], vmax, z10, tWeldGun;
		MoveL [[264.24,-890.45,-120.68],[0.253161,-0.649527,-0.664896,-0.268211],[-1,0,0,0],[9E+09,9E+09,9E+09,9E+09,9E+09,9E+09]], vmax, z10, tWeldGun;
		ArcLStart [[263.48,-888.99,-134.98],[0.221199,-0.661534,-0.676257,-0.2369],[-1,-1,0,0],[9E+09,9E+09,9E+09,9E+09,9E+09,9E+09]], v40, seam13, weld13\Weave:=weave1, fine, tWeldGun;
		ArcLEnd [[229.44,-889.20,-134.98],[0.221239,-0.661471,-0.676322,-0.23685],[-1,-1,0,0],[9E+09,9E+09,9E+09,9E+09,9E+09,9E+09]], v10, seam13, weld13\Weave:=weave1, fine, tWeldGun;
		MoveL [[221.59,-928.39,0.88],[0.253241,-0.64951,-0.664872,-0.268236],[-1,0,0,0],[9E+09,9E+09,9E+09,9E+09,9E+09,9E+09]], vmax, z10, tWeldGun;
		MoveL [[149.12,-928.38,0.88],[0.253244,-0.649508,-0.664873,-0.268237],[-1,0,0,0],[9E+09,9E+09,9E+09,9E+09,9E+09,9E+09]], vmax, z10, tWeldGun;
		MoveL [[172.54,-889.34,-116.50],[0.226503,-0.659767,-0.673922,-0.243381],[-1,0,0,0],[9E+09,9E+09,9E+09,9E+09,9E+09,9E+09]], vmax, z10, tWeldGun;
		ArcLStart [[165.23,-888.02,-135.78],[0.226573,-0.659687,-0.674025,-0.243247],[-1,0,0,0],[9E+09,9E+09,9E+09,9E+09,9E+09,9E+09]], v40, seam13, weld13\Weave:=weave1, fine, tWeldGun;
		ArcL [[147.83,-888.01,-135.78],[0.226571,-0.659686,-0.674028,-0.243242],[-1,0,0,0],[9E+09,9E+09,9E+09,9E+09,9E+09,9E+09]], v10, seam13, weld13\Weave:=weave1, z0, tWeldGun;
		ArcLEnd [[139.82,-877.64,-135.79],[0.226611,-0.659668,-0.674028,-0.243252],[-1,0,0,0],[9E+09,9E+09,9E+09,9E+09,9E+09,9E+09]], v10, seam13, weld13\Weave:=weave1, fine, tWeldGun;
		MoveL [[144.21,-880.62,-47.38],[0.226564,-0.659716,-0.673945,-0.243396],[-1,0,0,0],[9E+09,9E+09,9E+09,9E+09,9E+09,9E+09]], vmax, z10, tWeldGun;
		MoveJ [[133.84,-1301.69,-30.86],[0.241723,0.664636,-0.669792,0.226294],[-1,-1,-2,0],[9E+09,9E+09,9E+09,9E+09,9E+09,9E+09]], vmax, z10, tWeldGun;
		MoveL [[133.71,-1366.85,-106.53],[0.241894,0.664487,-0.669849,0.226378],[-1,-1,-2,0],[9E+09,9E+09,9E+09,9E+09,9E+09,9E+09]], vmax, z10, tWeldGun;
		ArcLStart [[130.25,-1367.99,-128.92],[0.241824,0.66459,-0.669787,0.226333],[-1,-1,-2,0],[9E+09,9E+09,9E+09,9E+09,9E+09,9E+09]], v40, seam13, weld13\Weave:=weave1, fine, tWeldGun;
		ArcL [[141.44,-1357.71,-129.71],[0.241825,0.664601,-0.669776,0.226332],[-1,-1,-2,0],[9E+09,9E+09,9E+09,9E+09,9E+09,9E+09]], v10, seam13, weld13\Weave:=weave1, z0, tWeldGun;
		ArcLEnd [[168.04,-1357.71,-129.70],[0.241826,0.664613,-0.669764,0.226333],[-1,0,-2,0],[9E+09,9E+09,9E+09,9E+09,9E+09,9E+09]], v10, seam13, weld13\Weave:=weave1, fine, tWeldGun;
		MoveL [[158.56,-1358.34,-123.52],[0.241852,0.664567,-0.669792,0.226359],[-1,0,-2,0],[9E+09,9E+09,9E+09,9E+09,9E+09,9E+09]], vmax, z10, tWeldGun;
		MoveL [[159.11,-1275.83,-114.78],[0.241858,0.66457,-0.669789,0.226353],[-1,0,-2,0],[9E+09,9E+09,9E+09,9E+09,9E+09,9E+09]], vmax, z10, tWeldGun;
		MoveJ [[258.04,-1277.97,58.89],[0.241847,0.664588,-0.669783,0.226327],[-1,0,-2,0],[9E+09,9E+09,9E+09,9E+09,9E+09,9E+09]], vmax, z10, tWeldGun;
		MoveL [[221.83,-1345.35,-107.31],[0.241807,0.664705,-0.66968,0.226331],[-1,0,-2,0],[9E+09,9E+09,9E+09,9E+09,9E+09,9E+09]], vmax, z10, tWeldGun;
		ArcLStart [[220.13,-1357.40,-129.80],[0.241823,0.664701,-0.669677,0.226336],[-1,0,-2,0],[9E+09,9E+09,9E+09,9E+09,9E+09,9E+09]], v40, seam13, weld13\Weave:=weave1, fine, tWeldGun;
		ArcLEnd [[267.51,-1357.98,-130.61],[0.241819,0.66468,-0.669702,0.226326],[-1,0,-2,0],[9E+09,9E+09,9E+09,9E+09,9E+09,9E+09]], v10, seam13, weld13\Weave:=weave1, fine, tWeldGun;
		MoveL [[258.91,-1359.32,-112.60],[0.241795,0.664688,-0.669704,0.226323],[-1,0,-2,0],[9E+09,9E+09,9E+09,9E+09,9E+09,9E+09]], vmax, z10, tWeldGun;
		MoveL [[334.62,-1358.15,-112.61],[0.241795,0.664695,-0.669698,0.22632],[-1,0,-2,0],[9E+09,9E+09,9E+09,9E+09,9E+09,9E+09]], vmax, z10, tWeldGun;
		ArcLStart [[338.01,-1358.74,-130.64],[0.232433,0.668117,-0.666401,0.235595],[-1,0,-2,0],[9E+09,9E+09,9E+09,9E+09,9E+09,9E+09]], v40, seam13, weld13\Weave:=weave1, fine, tWeldGun;
		ArcL [[380.78,-1359.35,-130.44],[0.232435,0.668122,-0.666396,0.235593],[-1,0,-2,0],[9E+09,9E+09,9E+09,9E+09,9E+09,9E+09]], v10, seam13, weld13\Weave:=weave1, z0, tWeldGun;
		ArcLEnd [[387.19,-1369.56,-130.08],[0.232406,0.668099,-0.666443,0.235554],[-1,0,-2,0],[9E+09,9E+09,9E+09,9E+09,9E+09,9E+09]], v10, seam13, weld13\Weave:=weave1, fine, tWeldGun;
		MoveL [[388.15,-1371.45,-115.55],[0.241783,0.664794,-0.669629,0.226246],[-1,0,-2,0],[9E+09,9E+09,9E+09,9E+09,9E+09,9E+09]], vmax, z10, tWeldGun;
		MoveL [[462.23,-1370.00,-115.57],[0.241782,0.664808,-0.669614,0.226252],[-1,0,-2,0],[9E+09,9E+09,9E+09,9E+09,9E+09,9E+09]], vmax, z10, tWeldGun;
		ArcLStart [[461.60,-1369.37,-129.68],[0.241783,0.664938,-0.669496,0.226215],[-1,0,-2,0],[9E+09,9E+09,9E+09,9E+09,9E+09,9E+09]], v40, seam13, weld13\Weave:=weave1, fine, tWeldGun;
		ArcL [[473.38,-1360.24,-130.12],[0.241808,0.664971,-0.669441,0.226257],[-1,0,-2,0],[9E+09,9E+09,9E+09,9E+09,9E+09,9E+09]], v10, seam13, weld13\Weave:=weave1, z0, tWeldGun;
		ArcL [[571.55,-1362.20,-130.09],[0.241802,0.66495,-0.669468,0.226244],[-1,0,-2,0],[9E+09,9E+09,9E+09,9E+09,9E+09,9E+09]], v10, seam13, weld13\Weave:=weave1, z0, tWeldGun;
		ArcLEnd [[580.07,-1371.37,-128.12],[0.24181,0.664943,-0.669481,0.226216],[-1,0,-2,0],[9E+09,9E+09,9E+09,9E+09,9E+09,9E+09]], v10, seam13, weld13\Weave:=weave1, fine, tWeldGun;
		MoveL [[580.73,-1368.76,-109.60],[0.211834,0.675038,-0.658294,0.257099],[-1,0,-2,0],[9E+09,9E+09,9E+09,9E+09,9E+09,9E+09]], vmax, z10, tWeldGun;
		MoveL [[580.72,-1333.23,219.73],[0.211837,0.67505,-0.658281,0.257098],[-1,0,-2,0],[9E+09,9E+09,9E+09,9E+09,9E+09,9E+09]], vmax, z10, tWeldGun;
		MoveJ [[285.51,-1411.06,96.42],[0.200981,-0.684372,-0.670688,-0.203517],[-1,-1,0,0],[9E+09,9E+09,9E+09,9E+09,9E+09,9E+09]], vmax, z10, tWeldGun;
		MoveL [[274.46,-1414.45,-119.52],[0.177177,-0.688252,-0.683971,-0.164625],[-1,-1,0,0],[9E+09,9E+09,9E+09,9E+09,9E+09,9E+09]], vmax, z10, tWeldGun;
		ArcLStart [[278.96,-1410.51,-127.90],[0.177207,-0.688228,-0.683996,-0.164593],[-1,-1,0,0],[9E+09,9E+09,9E+09,9E+09,9E+09,9E+09]], v40, seam13, weld13\Weave:=weave1, fine, tWeldGun;
		ArcLEnd [[343.75,-1409.54,-127.69],[0.17722,-0.688224,-0.683998,-0.164585],[-1,-1,0,0],[9E+09,9E+09,9E+09,9E+09,9E+09,9E+09]], v10, seam13, weld13\Weave:=weave1, fine, tWeldGun;
		MoveL [[345.60,-1413.44,-114.91],[0.177186,-0.688241,-0.683983,-0.164611],[-1,-1,0,0],[9E+09,9E+09,9E+09,9E+09,9E+09,9E+09]], vmax, z10, tWeldGun;
		MoveL [[346.19,-1405.53,-125.02],[0.247913,-0.667275,-0.663007,-0.231743],[-1,-1,0,0],[9E+09,9E+09,9E+09,9E+09,9E+09,9E+09]], vmax, z10, tWeldGun;
		ArcLStart [[346.19,-1405.93,-131.01],[0.24792,-0.667274,-0.663008,-0.231738],[-1,-1,0,0],[9E+09,9E+09,9E+09,9E+09,9E+09,9E+09]], v20, seam13, weld13\Weave:=weave1, fine, tWeldGun;
		ArcLEnd [[281.40,-1405.84,-130.04],[0.247958,-0.667273,-0.662986,-0.231764],[-1,-1,0,0],[9E+09,9E+09,9E+09,9E+09,9E+09,9E+09]], v10, seam13, weld13\Weave:=weave1, fine, tWeldGun;
		MoveL [[278.23,-1407.14,-118.05],[0.247851,-0.667236,-0.663096,-0.23167],[-1,-1,0,0],[9E+09,9E+09,9E+09,9E+09,9E+09,9E+09]], vmax, z10, tWeldGun;
		MoveJ [[748.76,-1435.11,122.90],[0.309636,-0.639534,-0.632199,-0.308944],[-1,0,0,0],[9E+09,9E+09,9E+09,9E+09,9E+09,9E+09]], vmax, z10, tWeldGun;
		MoveL [[747.76,-1423.09,122.93],[0.309631,-0.639515,-0.632217,-0.308951],[-1,0,0,0],[9E+09,9E+09,9E+09,9E+09,9E+09,9E+09]], vmax, z10, tWeldGun;
		ArcLStart [[746.39,-1409.34,121.28],[0.309822,-0.639514,-0.632123,-0.308955],[-1,0,0,0],[9E+09,9E+09,9E+09,9E+09,9E+09,9E+09]], v40, seam13, weld13\Weave:=weave1, fine, tWeldGun;
		ArcL [[756.39,-1410.13,113.73],[0.309845,-0.639542,-0.632066,-0.308991],[-1,0,0,0],[9E+09,9E+09,9E+09,9E+09,9E+09,9E+09]], v10, seam13, weld13\Weave:=weave1, z20, tWeldGun;
		ArcL [[758.90,-1409.80,105.35],[0.309852,-0.639538,-0.632076,-0.308971],[-1,0,0,0],[9E+09,9E+09,9E+09,9E+09,9E+09,9E+09]], v10, seam13, weld13\Weave:=weave1, z20, tWeldGun;
		ArcL [[763.61,-1409.23,93.16],[0.309915,-0.639536,-0.632081,-0.308902],[-1,0,0,0],[9E+09,9E+09,9E+09,9E+09,9E+09,9E+09]], v10, seam13, weld13\Weave:=weave1, z20, tWeldGun;
		ArcLEnd [[772.65,-1408.78,89.84],[0.327489,-0.630614,-0.623202,-0.326645],[-1,0,0,0],[9E+09,9E+09,9E+09,9E+09,9E+09,9E+09]], v10, seam13, weld13\Weave:=weave1, fine, tWeldGun;
		MoveL [[772.20,-1434.22,91.41],[0.309863,-0.63952,-0.632095,-0.30896],[-1,0,0,0],[9E+09,9E+09,9E+09,9E+09,9E+09,9E+09]], vmax, z10, tWeldGun;
		MoveL [[710.64,-1419.78,125.28],[0.30966,-0.639572,-0.632197,-0.308846],[-1,0,0,0],[9E+09,9E+09,9E+09,9E+09,9E+09,9E+09]], vmax, z10, tWeldGun;
		ArcLStart [[709.50,-1405.44,121.92],[0.309978,-0.63955,-0.63204,-0.308895],[-1,0,0,0],[9E+09,9E+09,9E+09,9E+09,9E+09,9E+09]], v40, seam13, weld13\Weave:=weave1, fine, tWeldGun;
		ArcL [[708.90,-1408.48,109.94],[0.309965,-0.639494,-0.632069,-0.308963],[-1,0,0,0],[9E+09,9E+09,9E+09,9E+09,9E+09,9E+09]], v10, seam13, weld13\Weave:=weave1, z10, tWeldGun;
		ArcLEnd [[694.10,-1408.36,88.68],[0.309922,-0.639534,-0.632102,-0.308856],[-1,0,0,0],[9E+09,9E+09,9E+09,9E+09,9E+09,9E+09]], v10, seam13, weld13\Weave:=weave1, fine, tWeldGun;
		MoveL [[694.77,-1422.13,93.38],[0.309744,-0.639622,-0.632095,-0.308866],[-1,0,0,0],[9E+09,9E+09,9E+09,9E+09,9E+09,9E+09]], vmax, z10, tWeldGun;
		MoveL [[627.48,-1417.65,-2.71],[0.30978,-0.639664,-0.632044,-0.308849],[-1,0,0,0],[9E+09,9E+09,9E+09,9E+09,9E+09,9E+09]], vmax, z10, tWeldGun;
		ArcLStart [[627.67,-1407.48,-6.35],[0.309842,-0.63961,-0.632098,-0.308786],[-1,0,0,0],[9E+09,9E+09,9E+09,9E+09,9E+09,9E+09]], v40, seam13, weld13\Weave:=weave1, fine, tWeldGun;
		ArcL [[595.68,-1406.53,-50.50],[0.309872,-0.63964,-0.632055,-0.308784],[-1,0,0,0],[9E+09,9E+09,9E+09,9E+09,9E+09,9E+09]], v10, seam13, weld13\Weave:=weave1, z0, tWeldGun;
		ArcLEnd [[545.26,-1406.30,-122.58],[0.309945,-0.639635,-0.63202,-0.308791],[-1,0,0,0],[9E+09,9E+09,9E+09,9E+09,9E+09,9E+09]], v10, seam13, weld13\Weave:=weave1, fine, tWeldGun;
		MoveL [[545.98,-1470.65,-122.68],[0.309529,-0.639772,-0.632153,-0.308653],[-1,0,0,0],[9E+09,9E+09,9E+09,9E+09,9E+09,9E+09]], vmax, z10, tWeldGun;
		MoveL [[546.01,-1470.74,261.49],[0.309463,-0.639811,-0.632171,-0.308601],[-1,0,0,0],[9E+09,9E+09,9E+09,9E+09,9E+09,9E+09]], vmax, z10, tWeldGun;
		MoveJ [[450.72,-1393.79,89.08],[0.00680651,0.918501,-0.0118982,0.395183],[-1,0,-3,0],[9E+09,9E+09,9E+09,9E+09,9E+09,9E+09]], vmax, z10, tWeldGun;
		MoveL [[571.40,-1393.78,20.15],[0.00679519,0.918514,-0.0118615,0.395152],[-1,0,-3,0],[9E+09,9E+09,9E+09,9E+09,9E+09,9E+09]], vmax, z10, tWeldGun;
		ArcLStart [[581.96,-1392.57,11.75],[0.00344146,0.944475,-0.0119614,0.328349],[-1,-1,-3,0],[9E+09,9E+09,9E+09,9E+09,9E+09,9E+09]], v50, seam13, weld13\Weave:=weave1, fine, tWeldGun;
		ArcLEnd [[582.10,-1373.59,11.74],[0.00343813,0.944488,-0.0119292,0.328313],[-1,-1,-3,0],[9E+09,9E+09,9E+09,9E+09,9E+09,9E+09]], v10, seam13, weld13\Weave:=weave1, fine, tWeldGun;
		MoveL [[564.04,-1375.65,36.36],[0.00687019,0.918524,-0.0118557,0.395129],[-1,0,-3,0],[9E+09,9E+09,9E+09,9E+09,9E+09,9E+09]], vmax, z10, tWeldGun;
		MoveJ [[280.70,-816.60,118.66],[0.243228,0.672922,-0.664156,0.216597],[-1,0,-2,0],[9E+09,9E+09,9E+09,9E+09,9E+09,9E+09]], vmax, z10, tWeldGun;
		MoveL [[280.25,-837.02,-125.82],[0.197071,0.688439,-0.669209,0.198433],[-1,0,-2,0],[9E+09,9E+09,9E+09,9E+09,9E+09,9E+09]], vmax, z10, tWeldGun;
		ArcLStart [[280.24,-840.38,-134.19],[0.197053,0.688439,-0.669224,0.1984],[-1,0,-2,0],[9E+09,9E+09,9E+09,9E+09,9E+09,9E+09]], v40, seam13, weld13\Weave:=weave1, fine, tWeldGun;
		ArcLEnd [[344.82,-841.20,-133.99],[0.197051,0.688474,-0.669184,0.198414],[-1,0,-2,0],[9E+09,9E+09,9E+09,9E+09,9E+09,9E+09]], v10, seam13, weld13\Weave:=weave1, fine, tWeldGun;
		MoveL [[342.48,-807.65,-103.06],[0.243058,0.673116,-0.664102,0.216347],[-1,0,-2,0],[9E+09,9E+09,9E+09,9E+09,9E+09,9E+09]], vmax, z10, tWeldGun;
		MoveL [[344.84,-838.46,-130.27],[0.239446,0.676384,-0.664309,0.209437],[-1,0,-2,0],[9E+09,9E+09,9E+09,9E+09,9E+09,9E+09]], v40, z10, tWeldGun;
		ArcLStart [[344.78,-844.07,-134.65],[0.239446,0.676419,-0.664275,0.209434],[-1,0,-2,0],[9E+09,9E+09,9E+09,9E+09,9E+09,9E+09]], v20, seam13, weld13\Weave:=weave1, fine, tWeldGun;
		ArcLEnd [[281.99,-843.61,-134.86],[0.239443,0.67643,-0.664266,0.20943],[-1,0,-2,0],[9E+09,9E+09,9E+09,9E+09,9E+09,9E+09]], v10, seam13, weld13\Weave:=weave1, fine, tWeldGun;
		MoveL [[282.15,-832.82,-127.25],[0.239444,0.676452,-0.664242,0.209434],[-1,0,-2,0],[9E+09,9E+09,9E+09,9E+09,9E+09,9E+09]], vmax, z10, tWeldGun;
		MoveL [[748.75,-833.29,121.02],[0.255044,0.669191,-0.660449,0.225708],[-1,0,-2,0],[9E+09,9E+09,9E+09,9E+09,9E+09,9E+09]], vmax, z10, tWeldGun;
		ArcLStart [[748.82,-845.27,116.40],[0.330396,0.607725,-0.646559,0.321669],[-1,-1,-2,0],[9E+09,9E+09,9E+09,9E+09,9E+09,9E+09]], v40, seam13, weld13\Weave:=weave1, fine, tWeldGun;
		ArcL [[755.03,-844.00,109.09],[0.290322,0.639723,-0.655361,0.277436],[-1,-1,-2,0],[9E+09,9E+09,9E+09,9E+09,9E+09,9E+09]], v10, seam13, weld13\Weave:=weave1, z10, tWeldGun;
		ArcL [[757.27,-844.12,99.83],[0.299668,0.635731,-0.648837,0.291645],[-1,-1,-2,0],[9E+09,9E+09,9E+09,9E+09,9E+09,9E+09]], v10, seam13, weld13\Weave:=weave1, z10, tWeldGun;
		ArcL [[759.23,-846.31,92.68],[0.324399,0.61002,-0.651776,0.312776],[-1,-1,-2,0],[9E+09,9E+09,9E+09,9E+09,9E+09,9E+09]], v10, seam13, weld13\Weave:=weave1, z10, tWeldGun;
		ArcLEnd [[771.00,-844.08,84.06],[0.302955,0.636757,-0.646551,0.291086],[-1,-1,-2,0],[9E+09,9E+09,9E+09,9E+09,9E+09,9E+09]], v10, seam13, weld13\Weave:=weave1, fine, tWeldGun;
		MoveL [[771.64,-817.13,91.59],[0.243124,0.673331,-0.663981,0.215974],[-1,0,-2,0],[9E+09,9E+09,9E+09,9E+09,9E+09,9E+09]], vmax, z10, tWeldGun;
		MoveL [[708.14,-831.16,119.68],[0.15545,0.696068,-0.587458,0.382384],[-1,0,-2,0],[9E+09,9E+09,9E+09,9E+09,9E+09,9E+09]], vmax, z10, tWeldGun;
		ArcLStart [[712.97,-843.74,118.07],[0.155383,0.69623,-0.587332,0.382309],[-1,0,-2,0],[9E+09,9E+09,9E+09,9E+09,9E+09,9E+09]], v40, seam13, weld13\Weave:=weave1, fine, tWeldGun;
		ArcL [[712.56,-843.72,109.06],[0.155377,0.696241,-0.587332,0.382295],[-1,0,-2,0],[9E+09,9E+09,9E+09,9E+09,9E+09,9E+09]], v10, seam13, weld13\Weave:=weave1, z10, tWeldGun;
		ArcLEnd [[698.15,-845.13,85.86],[0.155377,0.696295,-0.587271,0.382288],[-1,0,-3,0],[9E+09,9E+09,9E+09,9E+09,9E+09,9E+09]], v10, seam13, weld13\Weave:=weave1, fine, tWeldGun;
		MoveL [[695.84,-827.95,86.05],[0.15545,0.696101,-0.587428,0.382371],[-1,0,-3,0],[9E+09,9E+09,9E+09,9E+09,9E+09,9E+09]], vmax, z10, tWeldGun;
		MoveL [[627.64,-828.97,-7.49],[0.0770172,0.700241,-0.571715,0.420563],[-1,0,-3,0],[9E+09,9E+09,9E+09,9E+09,9E+09,9E+09]], vmax, z10, tWeldGun;
		ArcLStart [[633.67,-845.16,-6.28],[0.0770169,0.700292,-0.571642,0.420578],[-1,0,-3,0],[9E+09,9E+09,9E+09,9E+09,9E+09,9E+09]], v40, seam13, weld13\Weave:=weave1, fine, tWeldGun;
		ArcL [[596.83,-845.52,-57.04],[0.0770253,0.700303,-0.571621,0.420588],[-1,0,-3,0],[9E+09,9E+09,9E+09,9E+09,9E+09,9E+09]], v10, seam13, weld13\Weave:=weave1, z0, tWeldGun;
		ArcLEnd [[548.28,-846.01,-125.55],[0.0770081,0.700431,-0.571448,0.420612],[-1,0,-3,0],[9E+09,9E+09,9E+09,9E+09,9E+09,9E+09]], v10, seam13, weld13\Weave:=weave1, fine, tWeldGun;
		MoveL [[548.88,-773.40,234.33],[0.243177,0.673515,-0.663846,0.215757],[-1,0,-2,0],[9E+09,9E+09,9E+09,9E+09,9E+09,9E+09]], vmax, z10, tWeldGun;
		MoveJ [[554.61,-845.95,234.31],[0.0125503,-0.913958,0.00705174,-0.405554],[-1,0,-3,0],[9E+09,9E+09,9E+09,9E+09,9E+09,9E+09]], vmax, z10, tWeldGun;
		MoveL [[582.05,-856.11,17.60],[0.00387381,-0.924938,0.0107301,-0.379947],[-1,-1,-3,0],[9E+09,9E+09,9E+09,9E+09,9E+09,9E+09]], vmax, z10, tWeldGun;
		ArcLStart [[585.62,-857.53,7.43],[0.000905049,0.938079,-0.0234026,0.345629],[-1,-1,-3,0],[9E+09,9E+09,9E+09,9E+09,9E+09,9E+09]], v40, seam13, weld13\Weave:=weave1, fine, tWeldGun;
		ArcLEnd [[586.36,-878.74,9.84],[0.000872733,0.938089,-0.0233645,0.345607],[-1,-1,-3,0],[9E+09,9E+09,9E+09,9E+09,9E+09,9E+09]], v10, seam13, weld13\Weave:=weave1, fine, tWeldGun;
		MoveL [[536.09,-886.10,63.12],[0.0125865,-0.913974,0.00698526,-0.405519],[-1,0,-3,0],[9E+09,9E+09,9E+09,9E+09,9E+09,9E+09]], vmax, z10, tWeldGun;
		MoveJ [[730.00,-817.88,232.84],[0.157166,-0.839072,-0.35904,-0.37729],[-1,0,0,0],[9E+09,9E+09,9E+09,9E+09,9E+09,9E+09]], vmax, z10, tWeldGun;
		MoveL [[549.10,-773.76,241.36],[0.243257,0.673368,-0.663867,0.216061],[-1,0,2,0],[9E+09,9E+09,9E+09,9E+09,9E+09,9E+09]], vmax, z10, tWeldGun;
		MoveJ [[785.08,-1364.00,203.32],[0.00171317,-0.947718,0.00701896,-0.319029],[-1,-1,1,0],[9E+09,9E+09,9E+09,9E+09,9E+09,9E+09]], vmax, z10, tWeldGun;
		MoveL [[804.94,-1365.82,136.07],[0.00412652,-0.937645,0.00612413,-0.347517],[-1,-1,1,0],[9E+09,9E+09,9E+09,9E+09,9E+09,9E+09]], vmax, z10, tWeldGun;
		ArcLStart [[812.42,-1365.94,124.48],[0.00379784,0.946982,-0.00675814,0.321194],[-1,-1,1,0],[9E+09,9E+09,9E+09,9E+09,9E+09,9E+09]], v40, seam13, weld13\Weave:=weave1, fine, tWeldGun;
		ArcLEnd [[812.64,-1395.07,124.68],[0.003776,0.946976,-0.00683425,0.32121],[-1,-1,1,0],[9E+09,9E+09,9E+09,9E+09,9E+09,9E+09]], v10, seam13, weld13\Weave:=weave1, fine, tWeldGun;
		MoveL [[799.72,-1397.77,160.94],[0.00406041,-0.937645,0.00597838,-0.34752],[-1,-1,1,0],[9E+09,9E+09,9E+09,9E+09,9E+09,9E+09]], vmax, z10, tWeldGun;
		MoveJ [[912.45,-910.97,281.24],[0.471963,-0.00834501,-0.88125,-0.0240746],[-1,-1,-1,0],[9E+09,9E+09,9E+09,9E+09,9E+09,9E+09]], vmax, z10, tWeldGun;
		MoveL [[909.26,-887.50,143.89],[0.306131,-0.0105667,-0.951842,-0.0130303],[-1,0,-1,0],[9E+09,9E+09,9E+09,9E+09,9E+09,9E+09]], vmax, z10, tWeldGun;
		ArcLStart [[893.69,-886.11,123.81],[0.328979,-0.0104482,-0.944178,-0.0138978],[-1,0,-1,0],[9E+09,9E+09,9E+09,9E+09,9E+09,9E+09]], v40, seam13, weld13\Weave:=weave1, fine, tWeldGun;
		ArcLEnd [[893.41,-853.37,123.58],[0.329086,-0.0103992,-0.94414,-0.0139336],[-1,0,-1,0],[9E+09,9E+09,9E+09,9E+09,9E+09,9E+09]], v10, seam13, weld13\Weave:=weave1, fine, tWeldGun;
		MoveL [[912.81,-855.15,147.89],[0.30614,-0.0105141,-0.95184,-0.0129908],[-1,0,-1,0],[9E+09,9E+09,9E+09,9E+09,9E+09,9E+09]], vmax, z10, tWeldGun;
		MoveJ [[902.72,-1362.89,137.84],[0.306146,-0.0105253,-0.951838,-0.0129664],[-1,0,-1,0],[9E+09,9E+09,9E+09,9E+09,9E+09,9E+09]], vmax, z10, tWeldGun;
		MoveL [[906.45,-1364.21,149.51],[0.306018,-0.0106465,-0.951882,-0.0126526],[-1,0,-1,0],[9E+09,9E+09,9E+09,9E+09,9E+09,9E+09]], vmax, z10, tWeldGun;
		ArcLStart [[891.02,-1363.48,125.76],[0.312469,-0.0264928,-0.949412,-0.016711],[-1,0,-1,0],[9E+09,9E+09,9E+09,9E+09,9E+09,9E+09]], v40, seam13, weld13\Weave:=weave1, fine, tWeldGun;
		ArcLEnd [[890.86,-1394.28,125.74],[0.312487,-0.0264974,-0.949406,-0.0167219],[-1,0,-1,0],[9E+09,9E+09,9E+09,9E+09,9E+09,9E+09]], v10, seam13, weld13\Weave:=weave1, fine, tWeldGun;
		MoveL [[900.37,-1394.95,165.72],[0.306084,-0.0106333,-0.95186,-0.0127431],[-1,0,-1,0],[9E+09,9E+09,9E+09,9E+09,9E+09,9E+09]], vmax, z10, tWeldGun;
		MoveJ [[778.65,-875.76,193.58],[0.0091964,-0.885136,-0.0131126,-0.465058],[-1,0,1,0],[9E+09,9E+09,9E+09,9E+09,9E+09,9E+09]], vmax, z10, tWeldGun;
		MoveL [[804.53,-888.57,142.41],[0.00795263,-0.941332,-0.0147738,-0.337067],[-1,-1,1,0],[9E+09,9E+09,9E+09,9E+09,9E+09,9E+09]], vmax, z10, tWeldGun;
		!SingArea\Wrist;
		ArcLStart [[811.64,-888.32,124.05],[0.0114426,-0.956962,-0.0170149,-0.289488],[-1,-1,1,0],[9E+09,9E+09,9E+09,9E+09,9E+09,9E+09]], v40, seam13, weld13\Weave:=weave1, fine, tWeldGun;
		ArcLEnd [[811.66,-857.92,123.77],[0.0114433,-0.956965,-0.0170368,-0.289478],[-1,-1,1,0],[9E+09,9E+09,9E+09,9E+09,9E+09,9E+09]], v10, seam13, weld13\Weave:=weave1, fine, tWeldGun;
		MoveL [[808.29,-857.12,184.20],[0.00793204,-0.941309,-0.0148666,-0.337126],[-1,-1,1,0],[9E+09,9E+09,9E+09,9E+09,9E+09,9E+09]], vmax, z10, tWeldGun;
		MoveJ [[948.68,-756.38,498.60],[0.0965323,0.230115,0.963612,0.0958222],[-1,0,3,0],[9E+09,9E+09,9E+09,9E+09,9E+09,9E+09]], vmax, z10, tWeldGun;
		MoveJ [[889.29,-1470.79,212.85],[0.436349,-0.266701,-0.841159,-0.175847],[-1,-1,-1,0],[9E+09,9E+09,9E+09,9E+09,9E+09,9E+09]], vmax, z10, tWeldGun;
		MoveL [[894.09,-1534.28,133.14],[0.461389,-0.240587,-0.84872,-0.0944108],[-1,-1,-1,0],[9E+09,9E+09,9E+09,9E+09,9E+09,9E+09]], vmax, z10, tWeldGun;
		ArcLStart [[885.43,-1528.34,133.23],[0.461446,-0.240621,-0.848671,-0.094484],[-1,-1,-1,0],[9E+09,9E+09,9E+09,9E+09,9E+09,9E+09]], v20, seam13, weld13\Weave:=weave1, fine, tWeldGun;
		ArcLEnd [[885.61,-1527.74,82.82],[0.461461,-0.240633,-0.848659,-0.0944903],[-1,-1,-1,0],[9E+09,9E+09,9E+09,9E+09,9E+09,9E+09]], v10, seam13, weld13\Weave:=weave1, fine, tWeldGun;
		MoveL [[900.92,-1537.43,82.11],[0.461314,-0.240626,-0.848754,-0.0943692],[-1,-1,-1,0],[9E+09,9E+09,9E+09,9E+09,9E+09,9E+09]], vmax, z10, tWeldGun;
		MoveJ [[891.90,-1479.03,228.80],[0.436386,-0.266712,-0.841142,-0.175822],[-1,-1,-1,0],[9E+09,9E+09,9E+09,9E+09,9E+09,9E+09]], vmax, z10, tWeldGun;
		MoveJ [[806.64,-1540.34,222.36],[0.20159,-0.885065,-0.244063,-0.341256],[-1,-1,0,0],[9E+09,9E+09,9E+09,9E+09,9E+09,9E+09]], vmax, z10, tWeldGun;
		MoveL [[811.86,-1539.91,136.13],[0.138759,-0.782703,-0.30357,-0.525327],[-1,0,0,0],[9E+09,9E+09,9E+09,9E+09,9E+09,9E+09]], vmax, z10, tWeldGun;
		ArcLStart [[822.49,-1531.42,129.87],[0.138764,-0.782719,-0.303529,-0.525325],[-1,0,0,0],[9E+09,9E+09,9E+09,9E+09,9E+09,9E+09]], v20, seam13, weld13\Weave:=weave1, fine, tWeldGun;
		ArcLEnd [[822.42,-1530.63,81.75],[0.138811,-0.782749,-0.303569,-0.525244],[-1,0,0,0],[9E+09,9E+09,9E+09,9E+09,9E+09,9E+09]], v10, seam13, weld13\Weave:=weave1, fine, tWeldGun;
		MoveL [[728.99,-1561.34,83.75],[0.13874,-0.782769,-0.303661,-0.525181],[-1,0,0,0],[9E+09,9E+09,9E+09,9E+09,9E+09,9E+09]], vmax, z10, tWeldGun;
		MoveJ [[811.91,-1491.61,207.52],[0.234681,0.835234,-0.273321,0.415458],[-1,-1,1,0],[9E+09,9E+09,9E+09,9E+09,9E+09,9E+09]], vmax, z10, tWeldGun;
		MoveL [[824.61,-1496.30,152.68],[0.118504,0.727046,-0.62083,0.268201],[-1,0,2,0],[9E+09,9E+09,9E+09,9E+09,9E+09,9E+09]], vmax, z10, tWeldGun;
		ArcLStart [[819.47,-1510.90,147.25],[0.182482,0.780053,-0.515457,0.304175],[-1,0,2,0],[9E+09,9E+09,9E+09,9E+09,9E+09,9E+09]], v30, seam13, weld13\Weave:=weave1, fine, tWeldGun;
		ArcL [[837.40,-1500.49,149.54],[0.173112,0.785472,-0.518649,0.28995],[-1,0,2,0],[9E+09,9E+09,9E+09,9E+09,9E+09,9E+09]], v10, seam13, weld13\Weave:=weave1, z20, tWeldGun;
		ArcL [[855.15,-1500.28,148.72],[0.296293,0.614113,-0.713977,0.159098],[-1,-1,2,0],[9E+09,9E+09,9E+09,9E+09,9E+09,9E+09]], v10, seam13, weld13\Weave:=weave1, z20, tWeldGun;
		ArcLEnd [[876.79,-1513.20,143.98],[0.451866,0.277403,-0.841502,0.103639],[-1,-1,3,0],[9E+09,9E+09,9E+09,9E+09,9E+09,9E+09]], v10, seam13, weld13\Weave:=weave1, fine, tWeldGun;
		MoveL [[868.00,-1462.62,281.67],[0.305965,0.602072,-0.730191,0.103522],[-1,-1,2,0],[9E+09,9E+09,9E+09,9E+09,9E+09,9E+09]], vmax, z10, tWeldGun;
		SingArea\Wrist;
		MoveJ [[899.12,-810.48,249.50],[0.390921,-0.280842,-0.871961,-0.0894041],[-1,-1,-1,0],[9E+09,9E+09,9E+09,9E+09,9E+09,9E+09]], vmax, z10, tWeldGun;
		MoveL [[893.80,-750.95,157.22],[0.390907,-0.280846,-0.871963,-0.0894324],[-1,-1,-1,0],[9E+09,9E+09,9E+09,9E+09,9E+09,9E+09]], vmax, z10, tWeldGun;
		ArcLStart [[886.26,-737.00,144.61],[0.371803,-0.296755,-0.871375,-0.120018],[-1,-1,-1,0],[9E+09,9E+09,9E+09,9E+09,9E+09,9E+09]], v20, seam13, weld13\Weave:=weave1, fine, tWeldGun;
		ArcL [[867.13,-755.96,146.63],[0.285464,-0.473921,-0.811341,-0.188773],[-1,0,0,0],[9E+09,9E+09,9E+09,9E+09,9E+09,9E+09]], v10, seam13, weld13\Weave:=weave1, z20, tWeldGun;
		ArcL [[848.11,-757.28,148.84],[0.205831,-0.668254,-0.656615,-0.282713],[-1,-1,0,0],[9E+09,9E+09,9E+09,9E+09,9E+09,9E+09]], v10, seam13, weld13\Weave:=weave1, z20, tWeldGun;
		ArcLEnd [[828.37,-745.76,142.59],[0.175816,-0.825433,-0.409318,-0.346711],[-1,0,0,0],[9E+09,9E+09,9E+09,9E+09,9E+09,9E+09]], v10, seam13, weld13\Weave:=weave1, fine, tWeldGun;
		MoveL [[812.10,-741.27,179.87],[0.137944,-0.809833,-0.451489,-0.348283],[-1,-1,0,0],[9E+09,9E+09,9E+09,9E+09,9E+09,9E+09]], vmax, z10, tWeldGun;
		MoveJ [[813.33,-724.96,210.48],[0.173803,0.831678,-0.150908,0.505303],[-1,-1,1,0],[9E+09,9E+09,9E+09,9E+09,9E+09,9E+09]], vmax, z10, tWeldGun;
		MoveL [[811.73,-718.09,130.36],[0.235841,0.816262,-0.188511,0.492503],[-1,-1,2,0],[9E+09,9E+09,9E+09,9E+09,9E+09,9E+09]], vmax, z10, tWeldGun;
		ArcLStart [[819.21,-726.44,126.40],[0.272432,0.781687,-0.281297,0.485406],[-1,-1,2,0],[9E+09,9E+09,9E+09,9E+09,9E+09,9E+09]], v30, seam13, weld13\Weave:=weave1, fine, tWeldGun;
		ArcLEnd [[819.72,-727.92,70.71],[0.272443,0.781672,-0.281346,0.485396],[-1,-1,2,0],[9E+09,9E+09,9E+09,9E+09,9E+09,9E+09]], v10, seam13, weld13\Weave:=weave1, fine, tWeldGun;
		MoveL [[803.23,-727.44,244.82],[0.235868,0.816204,-0.188598,0.492553],[-1,-1,2,0],[9E+09,9E+09,9E+09,9E+09,9E+09,9E+09]], vmax, z10, tWeldGun;
		MoveJ [[895.52,-726.75,204.33],[0.55971,0.12946,-0.779061,0.251057],[-1,-1,3,0],[9E+09,9E+09,9E+09,9E+09,9E+09,9E+09]], vmax, z10, tWeldGun;
		MoveL [[895.52,-726.76,138.36],[0.559707,0.129464,-0.77906,0.251065],[-1,-1,3,0],[9E+09,9E+09,9E+09,9E+09,9E+09,9E+09]], v1000, z10, tWeldGun;
		ArcLStart [[880.65,-721.03,126.17],[0.534736,0.248309,-0.803914,0.0782544],[-1,-1,3,0],[9E+09,9E+09,9E+09,9E+09,9E+09,9E+09]], v30, seam13, weld13\Weave:=weave1, fine, tWeldGun;
		ArcLEnd [[882.61,-722.35,72.45],[0.534602,0.24832,-0.803987,0.0783806],[-1,-1,3,0],[9E+09,9E+09,9E+09,9E+09,9E+09,9E+09]], v10, seam13, weld13\Weave:=weave1, fine, tWeldGun;
		MoveL [[912.72,-716.39,263.71],[0.608762,0.242985,-0.747557,0.107361],[-1,-1,3,0],[9E+09,9E+09,9E+09,9E+09,9E+09,9E+09]], v1000, z10, tWeldGun;
		MoveJ [[948.69,-756.28,305.80],[0.0965088,0.229982,0.963647,0.0958049],[-1,1,2,0],[9E+09,9E+09,9E+09,9E+09,9E+09,9E+09]], vmax, z10, tWeldGun;
		MoveL [[867.49,-768.47,166.72],[0.130888,0.213603,0.942025,0.223231],[-1,1,2,0],[9E+09,9E+09,9E+09,9E+09,9E+09,9E+09]], vmax, z10, tWeldGun;
		ArcLStart [[867.89,-761.29,155.52],[0.130893,0.213602,0.942022,0.22324],[-1,1,2,0],[9E+09,9E+09,9E+09,9E+09,9E+09,9E+09]], v20, seam13, weld13\Weave:=weave1, fine, tWeldGun;
		ArcLEnd [[868.22,-847.27,156.47],[0.0965045,0.230044,0.963629,0.0958446],[-1,1,2,0],[9E+09,9E+09,9E+09,9E+09,9E+09,9E+09]], v10, seam13, weld13\Weave:=weave1, fine, tWeldGun;
		MoveL [[869.04,-847.26,165.53],[0.0964995,0.230018,0.963638,0.0958261],[-1,1,2,0],[9E+09,9E+09,9E+09,9E+09,9E+09,9E+09]], vmax, z10, tWeldGun;
		MoveL [[869.02,-913.92,164.66],[0.0964814,0.23003,0.963636,0.0958326],[-1,1,2,0],[9E+09,9E+09,9E+09,9E+09,9E+09,9E+09]], vmax, z10, tWeldGun;
		ArcLStart [[868.15,-911.68,158.53],[0.141521,0.205375,0.923592,0.291154],[-1,1,2,0],[9E+09,9E+09,9E+09,9E+09,9E+09,9E+09]], v10, seam13, weld13\Weave:=weave1, fine, tWeldGun;
		ArcLEnd [[867.65,-1009.97,158.58],[0.13854,0.205254,0.922447,0.29626],[-1,1,2,0],[9E+09,9E+09,9E+09,9E+09,9E+09,9E+09]], v10, seam13, weld13\Weave:=weave1, fine, tWeldGun;
		MoveL [[868.22,-1009.37,164.73],[0.0964767,0.230052,0.96363,0.0958467],[-1,1,2,0],[9E+09,9E+09,9E+09,9E+09,9E+09,9E+09]], vmax, z10, tWeldGun;
		MoveL [[868.20,-1076.23,165.04],[0.0964671,0.230068,0.963626,0.0958598],[-1,1,2,0],[9E+09,9E+09,9E+09,9E+09,9E+09,9E+09]], vmax, z10, tWeldGun;
		ArcLStart [[867.88,-1076.23,159.23],[0.143149,0.202435,0.916454,0.314072],[-1,0,2,0],[9E+09,9E+09,9E+09,9E+09,9E+09,9E+09]], v10, seam13, weld13\Weave:=weave1, fine, tWeldGun;
		ArcLEnd [[866.88,-1177.59,159.58],[0.143489,0.202315,0.91616,0.314852],[-1,0,2,0],[9E+09,9E+09,9E+09,9E+09,9E+09,9E+09]], v10, seam13, weld13\Weave:=weave1, fine, tWeldGun;
		MoveL [[867.42,-1177.54,165.19],[0.0964178,0.230045,0.963637,0.0958523],[-1,1,2,0],[9E+09,9E+09,9E+09,9E+09,9E+09,9E+09]], vmax, z10, tWeldGun;
		MoveL [[866.59,-1244.32,164.65],[0.0963764,0.230062,0.963637,0.09585],[-1,1,2,0],[9E+09,9E+09,9E+09,9E+09,9E+09,9E+09]], vmax, z10, tWeldGun;
		ArcLStart [[867.16,-1244.30,161.05],[0.207996,0.187449,0.925709,0.254292],[-1,1,2,0],[9E+09,9E+09,9E+09,9E+09,9E+09,9E+09]], v10, seam13, weld13\Weave:=weave1, fine, tWeldGun;
		ArcLEnd [[866.04,-1344.20,159.16],[0.143885,0.207692,0.924941,0.283981],[-1,0,2,0],[9E+09,9E+09,9E+09,9E+09,9E+09,9E+09]], v10, seam13, weld13\Weave:=weave1, fine, tWeldGun;
		MoveL [[866.50,-1344.41,165.64],[0.0963592,0.230099,0.963628,0.0958744],[-1,1,2,0],[9E+09,9E+09,9E+09,9E+09,9E+09,9E+09]], vmax, z10, tWeldGun;
		MoveL [[865.99,-1410.63,164.60],[0.0963345,0.230139,0.963618,0.0959015],[-1,0,2,0],[9E+09,9E+09,9E+09,9E+09,9E+09,9E+09]], vmax, z10, tWeldGun;
		ArcLStart [[861.54,-1420.22,162.47],[0.0725054,0.284795,0.912906,-0.283264],[-1,1,1,0],[9E+09,9E+09,9E+09,9E+09,9E+09,9E+09]], v10, seam13, weld13\Weave:=weave1, fine, tWeldGun;
		ArcLEnd [[861.20,-1513.68,162.90],[0.072529,0.284809,0.912877,-0.283336],[-1,1,1,0],[9E+09,9E+09,9E+09,9E+09,9E+09,9E+09]], v10, seam13, weld13\Weave:=weave1, fine, tWeldGun;
		MoveL [[866.02,-1496.51,276.55],[0.0655721,0.243738,0.945871,-0.204013],[-1,1,2,0],[9E+09,9E+09,9E+09,9E+09,9E+09,9E+09]], vmax, z10, tWeldGun;
		MoveL [[-51.14,-815.87,929.70],[0.371764,-0.594065,-0.605839,-0.376614],[-2,-1,3,0],[9E+09,9E+09,9E+09,9E+09,9E+09,9E+09]], vmax, z10, tWeldGun;
	ENDPROC
	PROC rRUNSide1A()
           	rTestPosTop;
		TPWrite "Side 1 A";
		MoveJ pSafeS1, vmax, fine, tWeldGun;
		!Code Goes Here
		MoveJ [[1195.77,967.47,624.34],[0.0211986,-0.292543,0.866333,0.404273],[0,-1,1,1],[9E+09,9E+09,9E+09,9E+09,9E+09,9E+09]], v1000, z20, tWeldGun;
		MoveJ [[1202.08,958.55,27.66],[0.0678226,-0.111826,0.895436,0.425548],[0,-1,0,1],[9E+09,9E+09,9E+09,9E+09,9E+09,9E+09]], v1000, z20, tWeldGun;
		!SingArea\Wrist;
		MoveL [[1208.05,954.10,-0.16],[0.135153,-0.0819853,0.912836,0.376488],[0,0,0,1],[9E+09,9E+09,9E+09,9E+09,9E+09,9E+09]], v1000, z5, tWeldGun;
		ArcLStart [[1208.06,965.49,-4.37],[0.135156,-0.0819687,0.912838,0.376485],[0,0,0,1],[9E+09,9E+09,9E+09,9E+09,9E+09,9E+09]], v5, seam13, weld13\Weave:=weave1, fine, tWeldGun;
		ArcLEnd [[1181.66,965.49,-4.39],[0.13515,-0.0819703,0.91284,0.376483],[0,0,0,1],[9E+09,9E+09,9E+09,9E+09,9E+09,9E+09]], v5, seam13, weld13\Weave:=weave1, fine, tWeldGun;
		MoveL [[1180.50,960.73,100.66],[0.067842,-0.111808,0.895423,0.425576],[0,-1,0,1],[9E+09,9E+09,9E+09,9E+09,9E+09,9E+09]], vmax, z0, tWeldGun;
		MoveL [[867.04,1014.85,67.84],[0.0692843,-0.0563275,0.92497,-0.369403],[0,1,-1,1],[9E+09,9E+09,9E+09,9E+09,9E+09,9E+09]], vmax, z0, tWeldGun;
		MoveL [[869.49,1011.42,-5.10],[0.0692967,-0.0563794,0.924948,-0.369448],[0,1,-1,1],[9E+09,9E+09,9E+09,9E+09,9E+09,9E+09]], vmax, z0, tWeldGun;
		ArcLStart [[866.09,1001.23,-5.72],[0.0692908,-0.0564024,0.924941,-0.369462],[0,1,-1,1],[9E+09,9E+09,9E+09,9E+09,9E+09,9E+09]], v5, seam13, weld13\Weave:=weave1, fine, tWeldGun;
		ArcLEnd [[888.69,1001.23,-5.74],[0.0692889,-0.056409,0.92494,-0.369464],[0,1,-1,1],[9E+09,9E+09,9E+09,9E+09,9E+09,9E+09]], v5, seam13, weld13\Weave:=weave1, fine, tWeldGun;
		MoveL [[886.66,1008.91,119.93],[0.0693309,-0.056349,0.924962,-0.369411],[0,1,-1,1],[9E+09,9E+09,9E+09,9E+09,9E+09,9E+09]], vmax, z0, tWeldGun;
		MoveL [[1179.30,1008.46,86.74],[0.107531,-0.15675,0.912414,-0.362448],[0,0,-1,1],[9E+09,9E+09,9E+09,9E+09,9E+09,9E+09]], vmax, z0, tWeldGun;
		MoveL [[1183.28,1011.87,-7.09],[0.107529,-0.156762,0.912406,-0.362464],[0,0,-1,1],[9E+09,9E+09,9E+09,9E+09,9E+09,9E+09]], vmax, z0, tWeldGun;
		ArcLStart [[1183.93,1004.55,-7.78],[0.11255,-0.153242,0.900123,-0.391955],[0,0,-1,1],[9E+09,9E+09,9E+09,9E+09,9E+09,9E+09]], v5, seam13, weld13\Weave:=weave1, fine, tWeldGun;
		ArcLEnd [[1208.23,1005.20,-7.81],[0.112533,-0.153252,0.900121,-0.391961],[0,0,-1,1],[9E+09,9E+09,9E+09,9E+09,9E+09,9E+09]], v5, seam13, weld13\Weave:=weave1, fine, tWeldGun;
		MoveL [[1201.20,1017.65,129.07],[0.213214,-0.193184,0.897426,-0.334435],[0,0,-1,1],[9E+09,9E+09,9E+09,9E+09,9E+09,9E+09]], vmax, z0, tWeldGun;
		MoveJ [[885.83,967.12,146.79],[0.0390937,-0.243498,0.889932,0.383668],[0,-1,0,1],[9E+09,9E+09,9E+09,9E+09,9E+09,9E+09]], vmax, z0, tWeldGun;
		MoveL [[883.03,960.85,-3.21],[0.0390774,-0.243493,0.88993,0.38368],[0,-1,0,1],[9E+09,9E+09,9E+09,9E+09,9E+09,9E+09]], vmax, z0, tWeldGun;
		ArcLStart [[885.43,969.37,-3.22],[0.032874,-0.244402,0.879946,0.406058],[0,-1,0,1],[9E+09,9E+09,9E+09,9E+09,9E+09,9E+09]], v5, seam13, weld13\Weave:=weave1, fine, tWeldGun;
		ArcLEnd [[863.05,968.77,-2.83],[0.0328735,-0.244393,0.879952,0.406051],[0,-1,0,1],[9E+09,9E+09,9E+09,9E+09,9E+09,9E+09]], v5, seam13, weld13\Weave:=weave1, fine, tWeldGun;
		MoveL [[862.21,949.49,214.06],[0.0424258,-0.242958,0.89504,0.371585],[0,-1,0,1],[9E+09,9E+09,9E+09,9E+09,9E+09,9E+09]], vmax, z0, tWeldGun;
		MoveL [[1197.39,1502.39,137.74],[0.0213351,-0.292247,0.866338,0.404469],[0,-1,0,1],[9E+09,9E+09,9E+09,9E+09,9E+09,9E+09]], vmax, z0, tWeldGun;
		MoveL [[1203.21,1507.85,-5.49],[0.0535985,-0.083673,0.917272,0.385667],[0,0,0,1],[9E+09,9E+09,9E+09,9E+09,9E+09,9E+09]], vmax, z0, tWeldGun;
		ArcLStart [[1208.84,1511.35,-6.24],[0.0869121,-0.0695749,0.91625,0.384827],[0,0,0,1],[9E+09,9E+09,9E+09,9E+09,9E+09,9E+09]], v5, seam13, weld13\Weave:=weave1, fine, tWeldGun;
		ArcLEnd [[1182.05,1511.56,-6.24],[0.0869119,-0.0695725,0.916249,0.38483],[0,0,0,1],[9E+09,9E+09,9E+09,9E+09,9E+09,9E+09]], v5, seam13, weld13\Weave:=weave1, fine, tWeldGun;
		MoveL [[1181.48,1503.16,158.48],[0.0212657,-0.292228,0.86634,0.404483],[0,-1,0,1],[9E+09,9E+09,9E+09,9E+09,9E+09,9E+09]], vmax, z0, tWeldGun;
		SingArea\Wrist;
		MoveL [[868.25,1555.51,187.44],[0.227112,-0.185081,0.888817,-0.352378],[0,1,-2,1],[9E+09,9E+09,9E+09,9E+09,9E+09,9E+09]], vmax, z0, tWeldGun;
		MoveL [[869.04,1559.86,-0.54],[0.159111,-0.150648,0.902234,-0.371434],[0,1,-2,1],[9E+09,9E+09,9E+09,9E+09,9E+09,9E+09]], vmax, z0, tWeldGun;
		ArcLStart [[868.80,1553.86,-11.63],[0.0826958,0.288816,-0.895527,0.328296],[0,1,-2,1],[9E+09,9E+09,9E+09,9E+09,9E+09,9E+09]], v5, seam13, weld13\Weave:=weave1, fine, tWeldGun;
		ArcLEnd [[890.38,1554.24,-11.26],[0.08271,0.28882,-0.895522,0.328302],[0,1,-2,1],[9E+09,9E+09,9E+09,9E+09,9E+09,9E+09]], v5, seam13, weld13\Weave:=weave1, fine, tWeldGun;
		MoveL [[888.12,1562.49,80.36],[0.227116,-0.185107,0.888791,-0.352426],[0,1,-2,1],[9E+09,9E+09,9E+09,9E+09,9E+09,9E+09]], vmax, z0, tWeldGun;
		MoveL [[1184.50,1555.09,41.59],[0.152145,-0.176338,0.927538,-0.292285],[0,1,-2,1],[9E+09,9E+09,9E+09,9E+09,9E+09,9E+09]], vmax, z0, tWeldGun;
		MoveL [[1187.22,1561.30,-0.15],[0.227083,-0.18512,0.888785,-0.352456],[0,0,-2,1],[9E+09,9E+09,9E+09,9E+09,9E+09,9E+09]], vmax, z0, tWeldGun;
		ArcLStart [[1176.88,1559.49,-13.57],[0.0395824,0.618604,-0.673706,0.402348],[0,1,-3,1],[9E+09,9E+09,9E+09,9E+09,9E+09,9E+09]], v5, seam13, weld13\Weave:=weave1, fine, tWeldGun;
		ArcLEnd [[1201.67,1559.48,-13.57],[0.0395886,0.618602,-0.673709,0.402344],[0,1,-3,1],[9E+09,9E+09,9E+09,9E+09,9E+09,9E+09]], v5, seam13, weld13\Weave:=weave1, fine, tWeldGun;
		MoveL [[1205.97,1566.31,170.25],[0.227077,-0.185152,0.88879,-0.352432],[0,0,-2,1],[9E+09,9E+09,9E+09,9E+09,9E+09,9E+09]], vmax, z0, tWeldGun;
		MoveL [[881.77,1504.38,147.85],[0.0212859,-0.292306,0.866337,0.404431],[0,-1,0,1],[9E+09,9E+09,9E+09,9E+09,9E+09,9E+09]], vmax, z0, tWeldGun;
		MoveL [[883.67,1496.64,-2.08],[0.003736,0.116344,0.927337,0.355663],[0,0,0,1],[9E+09,9E+09,9E+09,9E+09,9E+09,9E+09]], vmax, z0, tWeldGun;
		ArcLStart [[890.26,1508.62,-8.71],[0.00370307,0.116426,0.927317,0.355689],[0,0,0,1],[9E+09,9E+09,9E+09,9E+09,9E+09,9E+09]], v5, seam13, weld13\Weave:=weave1, fine, tWeldGun;
		ArcLEnd [[870.46,1508.84,-9.30],[0.00370904,0.116372,0.927332,0.355669],[0,0,0,1],[9E+09,9E+09,9E+09,9E+09,9E+09,9E+09]], v5, seam13, weld13\Weave:=weave1, fine, tWeldGun;
		MoveL [[865.68,1505.22,88.67],[0.0212437,-0.292287,0.866358,0.404403],[0,-1,0,1],[9E+09,9E+09,9E+09,9E+09,9E+09,9E+09]], vmax, z0, tWeldGun;
		MoveL [[42.29,1547.28,5.42],[0.0930027,-0.145662,0.911404,0.373466],[1,0,0,1],[9E+09,9E+09,9E+09,9E+09,9E+09,9E+09]], vmax, z0, tWeldGun;
		ArcLStart [[42.35,1556.28,-2.58],[0.0930041,-0.145652,0.911406,0.373465],[1,0,0,1],[9E+09,9E+09,9E+09,9E+09,9E+09,9E+09]], v5, seam13, weld13\Weave:=weave1, fine, tWeldGun;
		ArcLEnd [[12.16,1556.26,-2.62],[0.092997,-0.145631,0.911414,0.373455],[1,0,0,1],[9E+09,9E+09,9E+09,9E+09,9E+09,9E+09]], v5, seam13, weld13\Weave:=weave1, fine, tWeldGun;
		MoveL [[12.10,1550.46,9.38],[0.0929989,-0.14565,0.911414,0.373447],[1,0,0,1],[9E+09,9E+09,9E+09,9E+09,9E+09,9E+09]], vmax, z0, tWeldGun;
		MoveL [[-278.66,1557.62,11.31],[0.104661,-0.181311,0.91043,0.356779],[1,0,0,1],[9E+09,9E+09,9E+09,9E+09,9E+09,9E+09]], vmax, z0, tWeldGun;
		ArcLStart [[-279.68,1559.03,-0.89],[0.104654,-0.181325,0.910427,0.35678],[1,0,0,1],[9E+09,9E+09,9E+09,9E+09,9E+09,9E+09]], v5, seam13, weld13\Weave:=weave1, fine, tWeldGun;
		ArcLEnd [[-311.67,1559.02,-0.89],[0.104658,-0.181316,0.910428,0.35678],[1,0,0,1],[9E+09,9E+09,9E+09,9E+09,9E+09,9E+09]], v5, seam13, weld13\Weave:=weave1, fine, tWeldGun;
		MoveL [[-319.66,1562.55,534.71],[0.0907184,-0.623281,0.712938,0.30824],[1,0,0,1],[9E+09,9E+09,9E+09,9E+09,9E+09,9E+09]], vmax, z0, tWeldGun;
		MoveJ [[-204.06,743.62,410.35],[0.169831,0.702229,0.669586,-0.1723],[1,0,-2,0],[9E+09,9E+09,9E+09,9E+09,9E+09,9E+09]], vmax, z0, tWeldGun;
		MoveJ [[-336.86,555.26,14.49],[0.352891,0.90921,0.19794,-0.0981131],[0,0,-2,0],[9E+09,9E+09,9E+09,9E+09,9E+09,9E+09]], vmax, z0, tWeldGun;
		ArcLStart [[-336.82,549.96,7.35],[0.352834,0.909218,0.198016,-0.0980882],[0,0,-2,0],[9E+09,9E+09,9E+09,9E+09,9E+09,9E+09]], v5, seam13, weld13\Weave:=weave1, fine, tWeldGun;
		ArcLEnd [[-306.63,550.02,7.36],[0.352826,0.909225,0.197979,-0.0981254],[0,0,-2,0],[9E+09,9E+09,9E+09,9E+09,9E+09,9E+09]], v5, seam13, weld13\Weave:=weave1, fine, tWeldGun;
		MoveL [[-306.62,555.42,20.36],[0.352823,0.909224,0.197986,-0.0981282],[0,0,-2,0],[9E+09,9E+09,9E+09,9E+09,9E+09,9E+09]], vmax, z0, tWeldGun;
		MoveL [[-15.36,553.36,14.76],[0.325268,0.908092,0.244403,-0.0991795],[0,0,-2,0],[9E+09,9E+09,9E+09,9E+09,9E+09,9E+09]], vmax, z0, tWeldGun;
		ArcLStart [[-17.60,548.14,5.76],[0.325278,0.908086,0.244417,-0.0991689],[0,0,-2,0],[9E+09,9E+09,9E+09,9E+09,9E+09,9E+09]], v5, seam13, weld13\Weave:=weave1, fine, tWeldGun;
		ArcLEnd [[15.14,547.53,5.78],[0.325316,0.90808,0.244368,-0.0992218],[0,0,-2,0],[9E+09,9E+09,9E+09,9E+09,9E+09,9E+09]], v5, seam13, weld13\Weave:=weave1, fine, tWeldGun;
		MoveL [[16.53,551.56,14.73],[0.325268,0.908096,0.244389,-0.0991872],[0,0,-2,0],[9E+09,9E+09,9E+09,9E+09,9E+09,9E+09]], vmax, z0, tWeldGun;
		MoveL [[835.19,546.59,8.86],[0.354374,0.887507,0.294518,0.00309851],[0,-1,-2,0],[9E+09,9E+09,9E+09,9E+09,9E+09,9E+09]], vmax, z0, tWeldGun;
		ArcLStart [[835.20,539.59,0.06],[0.354373,0.887506,0.294524,0.00310593],[0,-1,-2,0],[9E+09,9E+09,9E+09,9E+09,9E+09,9E+09]], v5, seam13, weld13\Weave:=weave1, fine, tWeldGun;
		ArcLEnd [[863.20,539.59,0.06],[0.354375,0.887505,0.294525,0.00310201],[0,-1,-2,0],[9E+09,9E+09,9E+09,9E+09,9E+09,9E+09]], v5, seam13, weld13\Weave:=weave1, fine, tWeldGun;
		MoveL [[863.15,544.60,13.06],[0.354372,0.887507,0.29452,0.00310136],[0,-1,-2,0],[9E+09,9E+09,9E+09,9E+09,9E+09,9E+09]], vmax, z0, tWeldGun;
		ConfL\Off;
		MoveL [[1163.05,540.25,17.31],[0.272611,0.697866,0.657915,-0.0762502],[0,-1,-3,0],[9E+09,9E+09,9E+09,9E+09,9E+09,9E+09]], vmax, z0, tWeldGun;
		ArcLStart [[1163.07,535.25,2.31],[0.272614,0.697856,0.657925,-0.0762497],[0,-1,-3,0],[9E+09,9E+09,9E+09,9E+09,9E+09,9E+09]], v5, seam13, weld13\Weave:=weave1, fine, tWeldGun;
		ArcLEnd [[1194.26,535.80,2.30],[0.272634,0.697844,0.657929,-0.0762488],[0,-1,-3,0],[9E+09,9E+09,9E+09,9E+09,9E+09,9E+09]], v5, seam13, weld13\Weave:=weave1, fine, tWeldGun;
		MoveL [[1196.79,537.72,478.96],[0.266966,0.671404,0.686159,-0.0844522],[0,-1,-3,0],[9E+09,9E+09,9E+09,9E+09,9E+09,9E+09]], vmax, z10, tWeldGun;
		!MoveJ [[44.07,948.69,1172.83],[0.0459633,-0.688402,0.722614,0.0426485],[0,-1,0,0],[9E+09,9E+09,9E+09,9E+09,9E+09,9E+09]], vmax, z10, tWeldGun;
		MoveJ [[-340.94,933.57,290.70],[0.111592,-0.946666,-0.184924,-0.23911],[1,0,-2,0],[9E+09,9E+09,9E+09,9E+09,9E+09,9E+09]], vmax, z10, tWeldGun;
		MoveL [[-397.78,986.25,11.78],[0.351596,0.0366706,-0.934077,-0.0503611],[1,-1,-3,0],[9E+09,9E+09,9E+09,9E+09,9E+09,9E+09]], v1000, z1, tWeldGun;
		ArcLStart [[-403.49,989.79,-7.03],[0.351616,0.0366471,-0.934072,-0.0503412],[1,-1,-3,0],[9E+09,9E+09,9E+09,9E+09,9E+09,9E+09]], v5, seam13, weld13\Weave:=weave1, fine, tWeldGun;
		ArcL [[-403.49,967.40,-7.03],[0.351611,0.0366553,-0.934073,-0.0503411],[1,-1,-3,0],[9E+09,9E+09,9E+09,9E+09,9E+09,9E+09]], v5, seam13, weld13\Weave:=weave1, z1, tWeldGun;
		ArcLEnd [[-427.89,951.23,-5.19],[0.166204,-0.66206,-0.696086,-0.222527],[1,0,-2,0],[9E+09,9E+09,9E+09,9E+09,9E+09,9E+09]], v5, seam13, weld13\Weave:=weave1, fine, tWeldGun;
		MoveL [[-431.85,948.97,-5.89],[0.171367,-0.660865,-0.695544,-0.223854],[1,0,-2,0],[9E+09,9E+09,9E+09,9E+09,9E+09,9E+09]], vmax, z0, tWeldGun;
		MoveL [[-428.23,950.42,262.61],[0.171376,-0.660832,-0.695567,-0.223872],[1,0,2,0],[9E+09,9E+09,9E+09,9E+09,9E+09,9E+09]], vmax, z0, tWeldGun;
		MoveJ [[-1240.64,940.49,246.51],[0.200371,-0.594607,-0.764476,-0.147887],[1,0,2,0],[9E+09,9E+09,9E+09,9E+09,9E+09,9E+09]], vmax, z0, tWeldGun;
		MoveL [[-1260.68,943.74,-4.40],[0.21012,-0.673397,-0.681885,-0.193442],[1,0,2,0],[9E+09,9E+09,9E+09,9E+09,9E+09,9E+09]], v100, z0, tWeldGun;
		ArcLStart [[-1260.21,948.52,-5.98],[0.20711,-0.662828,-0.692164,-0.196656],[1,0,2,0],[9E+09,9E+09,9E+09,9E+09,9E+09,9E+09]], v5, seam13, weld13\Weave:=weave1, fine, tWeldGun;
		ArcL [[-1280.81,949.93,-3.17],[0.207115,-0.662841,-0.692149,-0.196661],[1,0,2,0],[9E+09,9E+09,9E+09,9E+09,9E+09,9E+09]], v5, seam13, weld13\Weave:=weave1, z1, tWeldGun;
		ArcLEnd [[-1285.17,976.24,-6.33],[0.116097,0.902245,0.0966076,0.403909],[1,0,3,0],[9E+09,9E+09,9E+09,9E+09,9E+09,9E+09]], v5, seam13, weld13\Weave:=weave1, fine, tWeldGun;
		MoveL [[-1282.96,979.96,80.63],[0.116018,0.902243,0.096661,0.403925],[1,0,3,0],[9E+09,9E+09,9E+09,9E+09,9E+09,9E+09]], vmax, z0, tWeldGun;
		MoveJ [[-1358.53,1155.99,133.80],[0.133739,0.955506,0.10811,0.239657],[1,0,3,0],[9E+09,9E+09,9E+09,9E+09,9E+09,9E+09]], vmax, z0, tWeldGun;
		MoveL [[-1353.88,1158.65,0.21],[0.0670978,0.939836,-0.00297634,0.33496],[1,0,3,0],[9E+09,9E+09,9E+09,9E+09,9E+09,9E+09]], vmax, z0, tWeldGun;
		ArcLStart [[-1346.23,1158.64,-6.27],[0.0671044,0.939837,-0.00297922,0.334957],[1,0,3,0],[9E+09,9E+09,9E+09,9E+09,9E+09,9E+09]], v5, seam13, weld13\Weave:=weave1, fine, tWeldGun;
		ArcL [[-1345.67,1179.98,-5.85],[0.0671069,0.939841,-0.00298187,0.334944],[1,0,3,0],[9E+09,9E+09,9E+09,9E+09,9E+09,9E+09]], v5, seam13, weld13\Weave:=weave1, z1, tWeldGun;
		ArcLEnd [[-1328.93,1191.80,-5.10],[0.263454,0.723647,-0.589037,0.244874],[1,0,4,0],[9E+09,9E+09,9E+09,9E+09,9E+09,9E+09]], v5, seam13, weld13\Weave:=weave1, fine, tWeldGun;
		MoveL [[-1328.99,1198.21,13.92],[0.263465,0.723639,-0.589044,0.244868],[1,0,4,0],[9E+09,9E+09,9E+09,9E+09,9E+09,9E+09]], v100, z0, tWeldGun;
		MoveL [[-1329.56,1242.98,151.23],[0.276586,0.758563,-0.567487,0.161373],[1,0,4,0],[9E+09,9E+09,9E+09,9E+09,9E+09,9E+09]], vmax, z0, tWeldGun;
		MoveJ [[-495.18,1248.58,261.21],[0.287177,0.742929,-0.58422,0.155801],[1,0,-1,0],[9E+09,9E+09,9E+09,9E+09,9E+09,9E+09]], vmax, z0, tWeldGun;
		MoveL [[-498.43,1199.39,-6.17],[0.287202,0.742915,-0.584226,0.155801],[1,0,-1,0],[9E+09,9E+09,9E+09,9E+09,9E+09,9E+09]], vmax, z0, tWeldGun;
		ArcLStart [[-490.85,1196.57,-6.80],[0.207313,0.685594,-0.661766,0.221468],[1,-1,0,0],[9E+09,9E+09,9E+09,9E+09,9E+09,9E+09]], v5, seam13, weld13\Weave:=weave1, fine, tWeldGun;
		ArcL [[-476.81,1196.58,-6.80],[0.207315,0.685597,-0.661764,0.221462],[1,-1,0,0],[9E+09,9E+09,9E+09,9E+09,9E+09,9E+09]], v5, seam13, weld13\Weave:=weave1, z1, tWeldGun;
		SingArea\Wrist;
		ArcLEnd [[-467.34,1165.99,-8.32],[0.359536,0.0381069,-0.931215,-0.0460599],[1,-1,1,0],[9E+09,9E+09,9E+09,9E+09,9E+09,9E+09]], v5, seam13, weld13\Weave:=weave1, fine, tWeldGun;
		MoveL [[-421.44,1139.09,130.73],[0.359544,0.0381675,-0.931204,-0.0461746],[1,-1,1,0],[9E+09,9E+09,9E+09,9E+09,9E+09,9E+09]], vmax, z0, tWeldGun;
		MoveJ [[-409.78,718.78,85.27],[0.233728,0.658735,-0.674888,0.236571],[1,-1,0,0],[9E+09,9E+09,9E+09,9E+09,9E+09,9E+09]], vmax, z0, tWeldGun;
		MoveL [[-411.03,718.90,-5.38],[0.233734,0.658739,-0.674886,0.236562],[1,-1,0,0],[9E+09,9E+09,9E+09,9E+09,9E+09,9E+09]], vmax, z0, tWeldGun;
		ArcLStart [[-411.03,713.89,-5.37],[0.233736,0.658741,-0.674882,0.236563],[1,-1,0,0],[9E+09,9E+09,9E+09,9E+09,9E+09,9E+09]], v5, seam13, weld13\Weave:=weave1, fine, tWeldGun;
		ArcLEnd [[-431.22,713.89,-5.37],[0.233731,0.658745,-0.674877,0.236572],[1,-1,0,0],[9E+09,9E+09,9E+09,9E+09,9E+09,9E+09]], v5, seam13, weld13\Weave:=weave1, fine, tWeldGun;
		MoveL [[-431.23,713.88,96.49],[0.233747,0.658736,-0.674884,0.236564],[1,-1,0,0],[9E+09,9E+09,9E+09,9E+09,9E+09,9E+09]], vmax, z0, tWeldGun;
		MoveL [[-1257.57,713.89,96.49],[0.233748,0.658741,-0.67488,0.236557],[1,-1,0,0],[9E+09,9E+09,9E+09,9E+09,9E+09,9E+09]], vmax, z0, tWeldGun;
		MoveL [[-1257.49,718.74,-3.31],[0.233762,0.658747,-0.674873,0.236549],[1,-1,0,0],[9E+09,9E+09,9E+09,9E+09,9E+09,9E+09]], vmax, z0, tWeldGun;
		ArcLStart [[-1259.46,713.99,-3.47],[0.233755,0.658769,-0.674854,0.23655],[1,-1,0,0],[9E+09,9E+09,9E+09,9E+09,9E+09,9E+09]], v5, seam13, weld13\Weave:=weave1, fine, tWeldGun;
		ArcLEnd [[-1282.29,713.74,-3.69],[0.233753,0.658786,-0.67484,0.236542],[1,-1,0,0],[9E+09,9E+09,9E+09,9E+09,9E+09,9E+09]], v5, seam13, weld13\Weave:=weave1, fine, tWeldGun;
		MoveL [[-1282.90,713.31,123.57],[0.233803,0.658736,-0.674861,0.236572],[1,-1,0,0],[9E+09,9E+09,9E+09,9E+09,9E+09,9E+09]], vmax, z0, tWeldGun;
		MoveJ [[-1344.23,1422.02,101.83],[0.226991,-0.675391,-0.661326,-0.234461],[1,0,-2,0],[9E+09,9E+09,9E+09,9E+09,9E+09,9E+09]], vmax, z0, tWeldGun;
		MoveL [[-1344.24,1422.02,-3.62],[0.226998,-0.675396,-0.66132,-0.234453],[1,0,-2,0],[9E+09,9E+09,9E+09,9E+09,9E+09,9E+09]], vmax, z0, tWeldGun;
		ArcLStart [[-1344.44,1428.64,-6.55],[0.226994,-0.67541,-0.661309,-0.234449],[1,0,-2,0],[9E+09,9E+09,9E+09,9E+09,9E+09,9E+09]], v5, seam13, weld13\Weave:=weave1, fine, tWeldGun;
		ArcLEnd [[-1324.68,1428.85,-6.59],[0.226993,-0.675407,-0.66131,-0.234455],[1,0,-2,0],[9E+09,9E+09,9E+09,9E+09,9E+09,9E+09]], v5, seam13, weld13\Weave:=weave1, fine, tWeldGun;
		MoveL [[-1320.89,1427.11,81.12],[0.226982,-0.675417,-0.661301,-0.234462],[1,0,-2,0],[9E+09,9E+09,9E+09,9E+09,9E+09,9E+09]], vmax, z0, tWeldGun;
		MoveL [[-494.97,1419.41,70.78],[0.226989,-0.675424,-0.661294,-0.234454],[1,0,-2,0],[9E+09,9E+09,9E+09,9E+09,9E+09,9E+09]], vmax, z0, tWeldGun;
		MoveL [[-494.98,1419.41,-5.90],[0.226987,-0.675436,-0.661284,-0.23445],[1,0,-2,0],[9E+09,9E+09,9E+09,9E+09,9E+09,9E+09]], vmax, z0, tWeldGun;
		ArcLStart [[-492.88,1429.57,-8.67],[0.226987,-0.675465,-0.661253,-0.234454],[1,0,-2,0],[9E+09,9E+09,9E+09,9E+09,9E+09,9E+09]], v5, seam13, weld13\Weave:=weave1, fine, tWeldGun;
		ArcLEnd [[-472.30,1429.32,-7.68],[0.226977,-0.675469,-0.661247,-0.234468],[1,0,-2,0],[9E+09,9E+09,9E+09,9E+09,9E+09,9E+09]], v5, seam13, weld13\Weave:=weave1, fine, tWeldGun;
		MoveL [[-196.11,1086.38,621.33],[0.226996,-0.675454,-0.661218,-0.234578],[1,0,-2,0],[9E+09,9E+09,9E+09,9E+09,9E+09,9E+09]], vmax, z0, tWeldGun;

		!code ends here

        MoveJ pSafeS1, vmax, z10, tWeldGun;
	ENDPROC



